// TwinCAT 3 PLC project LoadBank_Controller
// ProgramVersion: 3.1.4024.0
// libraries:
//   Tc2_Standard, * (Beckhoff Automation GmbH)
//   Tc2_System, * (Beckhoff Automation GmbH)
//   Tc2_Utilities, * (Beckhoff Automation GmbH)
//   Tc3_Module, * (Beckhoff Automation GmbH)
//   VisuSymbols,3.5.10.0,System
// project tree:
//   DUTs/ DUT_Alarm.TcDUT, DUT_Alarm_History_Record.TcDUT, DUT_Saved_Recipe.TcDUT, Recipe_Status.TcDUT, DUT_Emergency_Status.TcDUT, DUT_HMI_Step.TcDUT, DUT_Mode_Status.TcDUT, DUT_Recipe_Step.TcDUT, DUT_Simple_Config.TcDUT, DUT_Simple_Status.TcDUT
//   / GlobalTextList.TcGTLO, PlcTask.TcTTO, VisualizationManager.TcVMO (not stored), VISU_TASK.TcTTO
//   GVLs/ GVL_LoadBank_Constants.TcGVL, GVL_LoadBank_IO.TcGVL, GVL_LoadBank_Persistent.TcGVL, GVL_LoadBank_Runtime.TcGVL, GVL_Recipe_Storage.TcGVL
//   POUs/ FB_Auto_Mode.TcPOU, FB_DataLogger.TcPOU, FB_Gradual_Dump.TcPOU, FB_Alarm_Manager.TcPOU, FB_Load_Controller.TcPOU, FB_Maintenance_Mode.TcPOU, FB_Main_Contactor.TcPOU, FB_Manual_Mode.TcPOU, FB_Mode_Manager.TcPOU, FB_Numeric_Mode.TcPOU, FB_Recipe_Controller.TcPOU, FB_Recipe_Storage_Manager.TcPOU, FB_Reverse_Mode.TcPOU, FB_Single_Fan.TcPOU, FB_Temperature_Monitor.TcPOU, PRG_Main.TcPOU, PRG_Maint_Mode.TcPOU
// real-time tasks:
//   TASK PlcTask: cycle T#10ms, priority 20, ADS port 350
//   TASK VISU_TASK: cycle T#200000us, priority 30, ADS port 351

CONFIGURATION LoadBank_Controller
    RESOURCE PLC ON TwinCAT3
        TASK PlcTask(INTERVAL := T#10ms, PRIORITY := 20);
        TASK VISU_TASK(INTERVAL := T#200000us, PRIORITY := 30);
        PROGRAM PRG_Main WITH PlcTask : PRG_Main;
        PROGRAM VisuElems_Visu_Prg WITH VISU_TASK : VisuElems.Visu_Prg;
    END_RESOURCE
END_CONFIGURATION

// ---- DUTs/DUT_Alarm.TcDUT
// ============================================
// DUT_Alarm
// Structure for active alarm records
// ============================================

TYPE DUT_Alarm :
STRUCT
    ID                  : UINT;             // Alarm number (1-17)
    Name                : STRING(30);       // Short name "FAN FAULT"
    Description         : STRING(50);       // Detail "Motor overload tripped"
    Severity            : UINT;             // 1=Critical (Red), 2=Warning (Yellow)
    Active              : BOOL;             // Currently active?
    Acknowledged        : BOOL;             // Operator acknowledged?
    Timestamp_Occurred  : STRING(20);       // When alarm started
END_STRUCT
END_TYPE

// ---- DUTs/DUT_Alarm_History_Record.TcDUT
// ============================================
// DUT_Alarm_History_Record
// Structure for alarm history records
// ============================================

TYPE DUT_Alarm_History_Record :
STRUCT
    Alarm_ID            : UINT;             // Alarm number (1-17)
    Alarm_Name          : STRING(30);       // Short name
    Severity            : UINT;             // 1=Critical, 2=Warning
    Time_Occurred       : STRING(20);       // When alarm started
    Time_Cleared        : STRING(20);       // When alarm cleared
    Duration_Sec        : UDINT;            // How long active (seconds)
    Was_Acknowledged    : BOOL;             // Was it ack'd before clearing?
END_STRUCT
END_TYPE

// ---- DUTs/DUT_Saved_Recipe.TcDUT
// ============================================
// DATA TYPE: DUT_Saved_Recipe
// Add to your DUTs folder
// ============================================
TYPE DUT_Saved_Recipe :
STRUCT
    Recipe_Name             : STRING(40);       // Recipe display name
    Number_Of_Steps         : UINT;             // How many steps in this recipe
    Steps                   : ARRAY[1..20] OF DUT_Recipe_Step;  // The recipe steps
    Total_Duration          : TIME;             // Calculated total time
    Peak_Power_kW           : REAL;             // Calculated peak power
    Is_Valid                : BOOL;             // TRUE if recipe slot contains valid data
END_STRUCT
END_TYPE

// ---- DUTs/Recipe_Status.TcDUT
TYPE Recipe_Status :
STRUCT
    Recipe_Running          : BOOL;
    Recipe_Complete         : BOOL;
    Recipe_Aborted          : BOOL;
	Recipe_Paused 			: BOOL;
    Current_Step            : UINT;
    Current_Step_Name       : STRING(30);
    Current_Target_kW       : REAL;
    Step_Elapsed_Time       : TIME;
    Step_Remaining_Time     : TIME;
    Step_Duration           : TIME;
    Step_Progress_Pct       : REAL;
    Total_Recipe_Time       : TIME;
    Total_Elapsed_Time      : TIME;
    Total_Remaining_Time    : TIME;
    Recipe_Progress_Pct     : REAL;
    Status_Message          : STRING(100);
END_STRUCT
END_TYPE

// ---- DUTs/DUT_Emergency_Status.TcDUT
TYPE DUT_Emergency_Status :
STRUCT
    Emergency_Active        : BOOL;
    Emergency_Type          : STRING(20);
    Emergency_Complete      : BOOL;
    Ramp_Progress_Percent   : UINT;
    Status_Message          : STRING(100);
END_STRUCT
END_TYPE

// ---- DUTs/DUT_HMI_Step.TcDUT
TYPE DUT_HMI_Step :
STRUCT
    Step_Number             : UINT;
    Rated_Power_kW          : REAL;
    Status_Active           : BOOL;
    Status_Quarantined      : BOOL;
    Status_Feedback_Fault   : BOOL;
    Status_Power_Fault      : BOOL;
    Cycle_Count             : UDINT;
    Measured_Power_kW       : REAL;
    Power_Error_Percent     : REAL;
	Has_Feedback            : BOOL;
END_STRUCT
END_TYPE

// ---- DUTs/DUT_Mode_Status.TcDUT
TYPE DUT_Mode_Status :
STRUCT
    Active_Mode             : UINT;
    Mode_Name               : STRING(30);
    Mode_Ready              : BOOL;
    Mode_Transitioning      : BOOL;
    Status_Message          : STRING(100);
END_STRUCT
END_TYPE

// ---- DUTs/DUT_Recipe_Step.TcDUT
TYPE DUT_Recipe_Step :
STRUCT
    Step_Name               : STRING(40);
    Target_Power_kW         : REAL;
    Duration                : TIME;
    Enabled                 : BOOL := TRUE;
END_STRUCT
END_TYPE

// ---- DUTs/DUT_Simple_Config.TcDUT
TYPE DUT_Simple_Config :
STRUCT
    Number_Of_Steps         : UINT := 10;
    Number_Of_TCs           : UINT := 5;
    Rated_Voltage           : REAL := 480.0;
    Voltage_Name            : STRING(20) := '480V 3-Phase';
    Voltage_Tolerance       : REAL := 5.0;
    Step_Power              : ARRAY[1..100] OF REAL;
    Temp_Warning            : REAL := 80.0;
    Temp_Maximum            : REAL := 100.0;
    Temp_Critical           : REAL := 120.0;
    Temp_Dump_Rate          : REAL := 10.0;
    Fan_Pressurize_Time     : TIME := T#5s;
    Fan_Cooldown_Time       : TIME := T#30s;
    EStop_Controlled_Percent: REAL := 10.0;
    EStop_Controlled_Time   : TIME := T#1s;
    Auto_Level_Deadband     : REAL := 5.0;
    Step_Change_Delay       : TIME := T#500ms;
    Feedback_Timeout        : TIME := T#3s;
    Enable_Power_Monitoring : BOOL := TRUE;
    Power_Tolerance_Percent : REAL := 5.0;
    Power_Monitor_Delay     : TIME := T#10s;
END_STRUCT
END_TYPE

// ---- DUTs/DUT_Simple_Status.TcDUT
TYPE DUT_Simple_Status :
STRUCT
    Released_Power_kW       : REAL;
    Available_Power_kW      : REAL;
    Rated_Total_kW          : REAL;
    Power_Error_kW          : REAL;
    Active_Steps            : UINT;
    Quarantined_Steps       : UINT;
    Fan_Running             : BOOL;
    Fan_Fault               : BOOL;
    Fan_Cycle_Count         : UDINT;
    Temperature_Outlet_Avg  : REAL;
    Temperature_Outlet_Max  : REAL;
    Temperature_Inlet       : REAL;
    Temperature_DeltaT      : REAL;
    Hottest_TC_Number       : UINT;
    Voltage_L1_L2           : REAL;
    Voltage_L2_L3           : REAL;
    Voltage_L3_L1           : REAL;
    Voltage_Average         : REAL;
    Voltage_Imbalance       : REAL;
    Voltage_OK              : BOOL;
    Current_L1              : REAL;
    Current_L2              : REAL;
    Current_L3              : REAL;
    Current_Total           : REAL;
    Current_Imbalance       : REAL;
    System_Running          : BOOL;
    System_Ready            : BOOL;
    System_Fault            : BOOL;
    System_Warning          : BOOL;
    Emergency_Active        : BOOL;
    Temperature_Dump        : BOOL;
    Active_Mode             : UINT;
    Mode_Name               : STRING(30);
    Mode_Ready              : BOOL;
END_STRUCT
END_TYPE

// ---- GVLs/GVL_LoadBank_Constants.TcGVL
VAR_GLOBAL CONSTANT

    // ============================================
    // OPERATING MODES (ID numbers only)
    // ============================================
    LB_MODE_OFF             : UINT := 0;
    LB_MODE_AUTO_LEVELING   : UINT := 1;
    LB_MODE_NUMERIC    		: UINT := 2;
    LB_MODE_REVERSE_POWER   : UINT := 3;
    LB_MODE_MANUAL			: UINT := 4;
    LB_MODE_RECIPE          : UINT := 5;
    LB_MODE_MAINTENANCE     : UINT := 6;

    // ============================================
    // HARDWARE CONFIGURATION (Change per job)
    // ============================================
    LB_NUMBER_OF_STEPS      : UINT := 10;
    LB_NUMBER_OF_TCS        : UINT := 2;
    
    // ============================================
    // VOLTAGE CONFIGURATION
    // ============================================
    LB_VOLTAGE              : REAL := 480.0;
    LB_VOLTAGE_NAME         : STRING(20) := '480V 3-Phase';

    // ============================================
    // STEP POWER RATINGS (kW per step)
    // When you change LB_NUMBER_OF_STEPS, update this array to match
    // ============================================
    LB_STEP_POWER           : ARRAY[1..LB_NUMBER_OF_STEPS] OF REAL := [
        40.0, 40.0, 80.0, 80.0, 160.0, 160.0, 320.0, 320.0, 640.0, 640.0
    ];

    // ============================================
    // ARRAY LIMITS
    // ============================================
    LB_MAX_RECIPE_STEPS     : UINT := 20;
    LB_TREND_BUFFER_MAX     : UINT := 3600;
	
	// Manual Mode Switch Configuration
    LB_MANUAL_SWITCH_POWER      : ARRAY[1..8] OF REAL := [50.0, 100.0, 150.0, 200.0, 250.0, 300.0, 350.0, 400.0];
    LB_NUMBER_OF_SWITCHES       : USINT := 8;

END_VAR

// ---- GVLs/GVL_LoadBank_IO.TcGVL
VAR_GLOBAL

    // ============================================
    // EMERGENCY INPUTS (NC contacts)
    // TRUE = OK, FALSE = E-STOP PRESSED
    // ============================================
    IO_Emergency_Immediate      : BOOL;
    IO_Emergency_Controlled     : BOOL;

    // ============================================
    // MASTER ENABLE INPUT (Optional physical switch)
    // Only used when LB_ENABLE_PHYSICAL_MASTER = TRUE
    // ============================================
    IO_Physical_Master_Enable   : BOOL;

    // ============================================
    // FAN INPUTS
    // ============================================
    IO_Fan_Contactor_FB         : BOOL;             // NO: TRUE = contactor closed
    IO_Fan_Motor_Overload_OK    : BOOL;             // NC: TRUE = healthy, FALSE = FAULT
    IO_Fan_Pressure_OK          : BOOL;             // NO: TRUE = pressure OK

    // ============================================
    // MAIN CONTACTOR INPUT
    // ============================================
    IO_Main_Contactor_FB        : BOOL;             // NO: TRUE = contactor closed, load contactor

    // ============================================
    // LOAD STEP INPUTS
    // ============================================
    IO_Load_Contactor_FB        : ARRAY[1..LB_NUMBER_OF_STEPS] OF BOOL;     // NO: TRUE = closed
    IO_Step_Power               : ARRAY[1..LB_NUMBER_OF_STEPS] OF REAL;     // kW per step

    // ============================================
    // TEMPERATURE INPUTS
    // ============================================
    IO_Temperature_TC           : ARRAY[1..LB_NUMBER_OF_TCS] OF REAL;
    IO_Temperature_Inlet        : REAL;

    // ============================================
    // POWER METER INPUTS - VOLTAGE
    // ============================================
    IO_Voltage_L1_L2            : REAL;
    IO_Voltage_L2_L3            : REAL;
    IO_Voltage_L3_L1            : REAL;
    IO_Voltage_Average          : REAL;
    
    IO_Voltage_L1_LN            : REAL;
    IO_Voltage_L2_LN            : REAL;
    IO_Voltage_L3_LN            : REAL;

    // ============================================
    // POWER METER INPUTS - CURRENT
    // ============================================
    IO_Current_L1               : REAL;
    IO_Current_L2               : REAL;
    IO_Current_L3               : REAL;

    // ============================================
    // POWER METER INPUTS - SYSTEM
    // ============================================
    IO_Frequency                : REAL;
    IO_Power_Factor             : REAL;
    IO_Total_Power_kW           : REAL;
    IO_Total_Power_kVAR         : REAL;
    IO_Total_Power_kVA          : REAL;

    // ============================================
    // EXTERNAL POWER INPUT (Auto/Reverse modes)
    // ============================================
    IO_External_Power_kW        : REAL;

    // ============================================
    // DIGITAL OUTPUTS - CONTACTORS
    // ============================================
    IO_Fan_Contactor_Coil       : BOOL;
    IO_Main_Contactor_Coil      : BOOL;
    IO_Load_Contactor_Coil      : ARRAY[1..LB_NUMBER_OF_STEPS] OF BOOL;

    // ============================================
    // DIGITAL OUTPUTS - LED INDICATORS
    // ============================================
    IO_LED_General_Alarm        : BOOL;             // Red LED
    IO_LED_Warning              : BOOL;             // Yellow LED
    IO_LED_System_Normal        : BOOL;             // Green LED
	
	// ============================================
    // FAN PHYSICAL CONTROL (Optional)
    // Only used when LB_ENABLE_PHYSICAL_FAN = TRUE
    // ============================================
    IO_Physical_Fan_Start       : BOOL;             // Physical start button

END_VAR

// ---- GVLs/GVL_LoadBank_Persistent.TcGVL
// ============================================
// GVL_LoadBank_Persistent
// UPDATED: Separate EMG and TEMP dump settings
// ============================================

VAR_GLOBAL PERSISTENT

    // ============================================
    // TEMPERATURE CONFIG (ENG Page)
    // ============================================
    LB_OUTLET_WARNING_TEMP      : REAL := 350.0;
    LB_OUTLET_MAXIMUM_TEMP      : REAL := 400.0;
    LB_TC_OPEN_LIMIT            : REAL := 700.0;
    LB_TC_SHORT_LIMIT           : REAL := -50.0;
    
    LB_INLET_WARNING_TEMP       : REAL := 50.0;
    LB_INLET_MAXIMUM_TEMP       : REAL := 75.0;
    LB_INLET_TC_ENABLED         : BOOL := TRUE;

    // ============================================
    // FAN CONTROL (ENG Page)
    // ============================================
    LB_FAN_PRESSURIZE_TIME      : TIME := T#5s;
    LB_FAN_COOLDOWN_TIME        : TIME := T#180s;    // CHANGED: Was T#30s, now 3 min for normal/temp cooldown
    LB_FAN_FEEDBACK_TIMEOUT     : TIME := T#3s;
    LB_FAN_POST_DUMP_DELAY      : TIME := T#5s;      // CHANGED: Was T#3s, delay after EMG dump before fan stops
    LB_ENABLE_PHYSICAL_FAN      : BOOL := FALSE;

    // ============================================
    // MAIN CONTACTOR (ENG Page)
    // ============================================
    LB_MAIN_CONTACTOR_FB_TIMEOUT : TIME := T#3s;

    // ============================================
    // CONTROLLED EMERGENCY DUMP (ENG Page)
    // Fan uses short delay (LB_FAN_POST_DUMP_DELAY) after dump
    // ============================================
    LB_EMG_DUMP_PERCENT         : REAL := 10.0;     // NEW: % per step for EMG
    LB_EMG_DUMP_STEP_TIME       : TIME := T#1s;     // NEW: Time between steps for EMG

    // ============================================
    // OVER TEMPERATURE DUMP (ENG Page)
    // Fan uses full cooldown (LB_FAN_COOLDOWN_TIME) after dump
    // ============================================
    LB_TEMP_DUMP_PERCENT        : REAL := 10.0;     // NEW: % per step for temp
    LB_TEMP_DUMP_STEP_TIME      : TIME := T#2s;     // NEW: Time between steps for temp

    // ============================================
    // DUMP TIMEOUT (ENG Page)
    // ============================================
    LB_DUMP_TIMEOUT             : TIME := T#30s;    // KEPT: Safety timeout for any dump

    // ============================================
    // LOAD CONTROL
    // ============================================
    LB_AUTO_LEVEL_DEADBAND      : REAL := 5.0;
    LB_AUTO_LEVEL_HYSTERESIS    : REAL := 2.0;
    LB_STEP_UP_DELAY            : TIME := T#500ms;
    LB_STEP_DOWN_DELAY          : TIME := T#500ms;

    // ============================================
    // FEEDBACK MONITORING (ENG Page)
    // ============================================
    LB_ENABLE_FEEDBACK_MONITORING : BOOL := FALSE;
    LB_FEEDBACK_TIMEOUT           : TIME := T#3s;

    // ============================================
    // POWER MONITORING (ENG Page)
    // ============================================
    LB_ENABLE_POWER_MONITORING  : BOOL := FALSE;
    LB_POWER_TOLERANCE_PERCENT  : REAL := 5.0;
    LB_POWER_MONITOR_DELAY      : TIME := T#10s;

    // ============================================
    // VOLTAGE IMBALANCE (ENG Page)
    // ============================================
    LB_VOLTAGE_TOLERANCE        : REAL := 5.0;
    LB_V_IMBALANCE_WARNING      : REAL := 1.0;
    LB_V_IMBALANCE_CRITICAL     : REAL := 2.0;

    // ============================================
    // CURRENT IMBALANCE (ENG Page)
    // ============================================
    LB_I_IMBALANCE_WARNING      : REAL := 1.0;
    LB_I_IMBALANCE_CRITICAL     : REAL := 2.0;

    // ============================================
    // DATA LOGGER (ENG Page)
    // ============================================
    LB_LOG_ENABLE               : BOOL := TRUE;
    LB_USB_LOG_ENABLE           : BOOL := TRUE;
    LB_LOG_SAMPLE_TIME          : TIME := T#10s;
    LB_TREND_BUFFER_SIZE        : UINT := 360;
    LB_USB_LOG_PATH             : STRING(100) := 'C:\DataLog\';

    // ============================================
    // HMI DISPLAY CONFIG (ENG Page)
    // ============================================
    LB_HMI_Config_Mode_Auto     : BOOL := TRUE;
    LB_HMI_Config_Mode_Reverse  : BOOL := FALSE;
    LB_HMI_Config_Mode_Manual   : BOOL := FALSE;

    // ============================================
    // HMI THEME (Customer Page)
    // ============================================
    LB_HMI_Dark_Mode            : BOOL := FALSE;

    // ============================================
    // MAINTENANCE (Customer Page)
    // ============================================
    LB_Maint_Test_Duration_Sec  : INT := 30;
    
    // ============================================
    // MASTER ENABLE CONFIG (ENG Page)
    // ============================================
    LB_ENABLE_PHYSICAL_MASTER   : BOOL := FALSE;
    
    // ============================================
    // Engineer Login Credentials
    // ============================================
    HMI_Eng_Username        : STRING(20) := 'eng';
    HMI_Eng_Password        : STRING(20) := 'loadbank2025';
    HMI_Eng_Timeout_Min     : INT := 10;
	
	// Settings
	Maint_Mode_Power_Tolerance_Percent  : REAL := 10.0;
	Maint_Mode_Feedback_Timeout_ms      : INT := 2000;
	Maint_Mode_Test_Duration_Sec        : INT := 5;

END_VAR

// ---- GVLs/GVL_LoadBank_Runtime.TcGVL
// ============================================
// GVL_LoadBank_Runtime
// UPDATED: Added HMI status text variables
// ============================================

VAR_GLOBAL

    // ============================================
    // MASTER ENABLE CONTROL
    // ============================================
    HMI_Master_Enable           : BOOL;
    Master_Enable               : BOOL;
    Master_Enable_Blocked       : BOOL;
    Master_Enable_Was_Off       : BOOL;

    // ============================================
    // FAN START CONTROL
    // ============================================
    HMI_Fan_Start               : BOOL;
    Fan_Start_Command           : BOOL;
    Fan_Start_Blocked           : BOOL;
    Fan_Start_Was_Off           : BOOL;

    // ============================================
    // HMI MODE INPUTS
    // ============================================
    HMI_Mode_Select             : UINT;
    HMI_Target_Power_kW         : REAL;
    HMI_Target_Frequency        : REAL := 60.0;
    HMI_Target_Reverse_kW       : REAL;
    HMI_Recipe_Start            : BOOL;
    HMI_Recipe_Stop             : BOOL;
    HMI_Recipe_Pause            : BOOL;
    HMI_Manual_Step_Cmd         : ARRAY[1..LB_NUMBER_OF_STEPS] OF BOOL;
    HMI_Reset_Cmd               : BOOL;
    
    // ============================================
    // NUMERIC MODE HMI
    // ============================================
    Numeric_Mode_Status         : STRING(100);

    // ============================================
    // AUTO MODE HMI
    // ============================================
    HMI_Min_Load_kW             : REAL;
    Auto_Mode_Power_Error       : REAL;
    Auto_Mode_Status            : STRING(100);

    // ============================================
    // QUARANTINE CONTROL
    // ============================================
    Step_Quarantined            : ARRAY[1..LB_NUMBER_OF_STEPS] OF BOOL;
    Step_Quarantine_Feedback    : ARRAY[1..LB_NUMBER_OF_STEPS] OF BOOL;
    Step_Quarantine_Manual      : ARRAY[1..LB_NUMBER_OF_STEPS] OF BOOL;
    Step_Unquarantine_Cmd       : ARRAY[1..LB_NUMBER_OF_STEPS] OF BOOL;
    Step_Cycle_Count            : ARRAY[1..LB_NUMBER_OF_STEPS] OF UDINT;

    // ============================================
    // DUMP STATUS
    // ============================================
    Dump_Active                 : BOOL;
    Dump_Percent                : REAL := 100.0;
    Dump_Complete               : BOOL;
    Is_Temperature_Dump         : BOOL;
    Is_Emergency_Dump           : BOOL;

    // ============================================
    // MAIN CONTACTOR STATUS
    // ============================================
    Main_Contactor_Closed       : BOOL;
    Main_Contactor_Fault        : BOOL;
    Main_Contactor_Allowed      : BOOL;

    // ============================================
    // SYSTEM STATUS FLAGS
    // ============================================
    System_Ready                : BOOL;
    System_Running              : BOOL;
    System_Fault                : BOOL;

    // ============================================
    // ALARM STATUS
    // ============================================
    General_Alarm               : BOOL;
    General_Warning             : BOOL;
    System_Normal               : BOOL;
    Any_Fault_Active            : BOOL;

    // ============================================
    // ALARM COMMANDS (from HMI)
    // ============================================
    Alarm_Acknowledge_Cmd       : BOOL;
    Alarm_Reset_Cmd             : BOOL;

    // ============================================
    // STATUS TEXT (for HMI display)
    // ============================================
    Status_Fan                  : STRING(100);
    Status_Temperature          : STRING(100);
    Status_Main_Contactor       : STRING(100);
    Status_Load                 : STRING(100);
    Status_Dump                 : STRING(100);

    // ============================================
    // HMI STATUS BAR TEXT (NEW)
    // ============================================
    HMI_System_Status_Text      : STRING(100);      // NEW: Main status message for HMI status bar
    HMI_Alarm_Detail_Text       : STRING(100);      // NEW: Secondary detail message for HMI

    // ============================================
    // MODE CONTROL
    // ============================================
    Mode_Current                : UINT;
    Mode_Requested              : UINT;
    Mode_Target_Power           : REAL;

    // ============================================
    // IMBALANCE CALCULATIONS
    // ============================================
    Voltage_Imbalance_Percent   : REAL;
    Current_Imbalance_Percent   : REAL;
    Voltage_Imbalance_Warning   : BOOL;
    Voltage_Imbalance_Critical  : BOOL;
    Current_Imbalance_Warning   : BOOL;
    Current_Imbalance_Critical  : BOOL;

    // ============================================
    // TREND BUFFERS (for HMI)
    // ============================================
    Trend_Power_Released        : ARRAY[1..LB_TREND_BUFFER_MAX] OF REAL;
    Trend_Power_Target          : ARRAY[1..LB_TREND_BUFFER_MAX] OF REAL;
    Trend_Temp_TC1              : ARRAY[1..LB_TREND_BUFFER_MAX] OF REAL;
    Trend_Temp_TC2              : ARRAY[1..LB_TREND_BUFFER_MAX] OF REAL;
    Trend_Temp_TC3              : ARRAY[1..LB_TREND_BUFFER_MAX] OF REAL;
    Trend_Temp_TC4              : ARRAY[1..LB_TREND_BUFFER_MAX] OF REAL;
    Trend_Voltage_L1L2          : ARRAY[1..LB_TREND_BUFFER_MAX] OF REAL;
    Trend_Voltage_L2L3          : ARRAY[1..LB_TREND_BUFFER_MAX] OF REAL;
    Trend_Voltage_L3L1          : ARRAY[1..LB_TREND_BUFFER_MAX] OF REAL;
    Trend_Current_I1            : ARRAY[1..LB_TREND_BUFFER_MAX] OF REAL;
    Trend_Current_I2            : ARRAY[1..LB_TREND_BUFFER_MAX] OF REAL;
    Trend_Current_I3            : ARRAY[1..LB_TREND_BUFFER_MAX] OF REAL;
    Trend_Index                 : UINT;
    Trend_Sample_Count          : UINT;

    // ============================================
    // SYSTEM STATUS STRUCT (for HMI)
    // ============================================
    LB_System_Status            : DUT_Simple_Status;
    LB_Mode_Status              : DUT_Mode_Status;
    LB_Emergency_Status         : DUT_Emergency_Status;
    LB_Recipe_Status            : Recipe_Status;

    // ============================================
    // STEP STATUS (for HMI)
    // ============================================
    LB_HMI_Steps                : ARRAY[1..LB_NUMBER_OF_STEPS] OF DUT_HMI_Step;
    LB_RATED_KW                 : ARRAY[1..LB_NUMBER_OF_STEPS] OF REAL;

    // ============================================
    // HMI HELPER VARIABLES
    // ============================================
    LB_HMI_Temperature_Status   : INT;
    LB_HMI_Fan_Status           : INT;
    LB_HMI_System_Status        : INT;
    LB_HMI_V_Imbalance_Status   : INT;
    LB_HMI_I_Imbalance_Status   : INT;

    LB_HMI_Released_Percent     : REAL;
    LB_HMI_Available_Percent    : REAL;

    LB_HMI_Active_Count         : INT;
    LB_HMI_Inactive_Count       : INT;
    LB_HMI_Quarantined_Count    : INT;
    LB_HMI_Total_Steps          : INT;

    LB_HMI_Active_Bar_Width     : REAL;
    LB_HMI_Inactive_Bar_Width   : REAL;
    LB_HMI_Quarantine_Bar_Width : REAL;

    LB_HMI_Hottest_TC           : INT;
    LB_HMI_Mode_Text            : STRING(20);
    LB_HMI_Mode_Ready           : BOOL;
    LB_HMI_Emergency_Text       : STRING(30);
    
    // ============================================
    // MANUAL MODE HMI (8 Switches)
    // ============================================
    HMI_Manual_Switch           : ARRAY[1..8] OF BOOL;
    HMI_Manual_Selected_kW      : REAL;
    Manual_Mode_Status          : STRING(100);
    
    // ============================================
    // RECIPE MODE HMI 
    // ============================================
    HMI_Recipe_Number_Of_Steps  : UINT := 5;
    HMI_Recipe_Steps            : ARRAY[1..20] OF DUT_Recipe_Step;
    
    // ============================================
    // REVERSE MODE HMI
    // ============================================
    HMI_Follow_Percentage       : REAL := 100.0;
    Reverse_Mode_Target_Power   : REAL;
    Reverse_Mode_Status         : STRING(100);
	
	// ============================================
    // ALARM MANAGER OUTPUTS (from FB_Alarm_Manager)
    // ============================================
    LB_Alarm_List               : ARRAY[1..20] OF DUT_Alarm;        // Active alarm list for HMI
    LB_Alarm_List_Count         : UINT;                              // Number of active alarms
    LB_Alarm_History            : ARRAY[1..50] OF DUT_Alarm_History_Record;  // History buffer
    LB_Alarm_History_Count      : UINT;                              // Number of history records
    
    LB_Critical_Alarm_Count     : UINT;                              // Critical alarm count
    LB_Warning_Count            : UINT;                              // Warning count
    LB_Total_Alarm_Count        : UINT;                              // Total active count
    LB_Unacknowledged_Count     : UINT;                              // Unacknowledged count
    
    LB_New_Alarm_Trigger        : BOOL;                              // Pulse for new alarm popup
    LB_Newest_Alarm_ID          : UINT;                              // ID of newest alarm
    LB_Newest_Alarm_Name        : STRING(30);                        // Name of newest alarm
    
    // ============================================
    // ALARM MANAGER COMMANDS (from HMI)
    // ============================================
    HMI_Alarm_Acknowledge       : ARRAY[1..20] OF BOOL;              // Acknowledge individual alarm
    HMI_Alarm_Acknowledge_All   : BOOL;                              // Acknowledge all alarms
    HMI_Alarm_Clear_History     : BOOL;                              // Clear history buffer
	
	// ============================================
// MAINTENANCE MODE HMI
// ============================================
// Commands (from HMI buttons)
Maint_Mode_Toggle_Fan               : BOOL;
Maint_Mode_Toggle_Step              : BOOL;
Maint_Mode_Reset_Test               : BOOL;
Maint_Mode_Selected_Step            : INT := 1;
Maint_Mode_Self_Test_Start          : BOOL;
Maint_Mode_Self_Test_Stop           : BOOL;


// Status (to HMI display)
Maint_Mode_Feedback_Match           : BOOL;
Maint_Mode_Response_Time_ms         : INT;
Maint_Mode_Power_Within_Tolerance   : BOOL;
Maint_Mode_Self_Test_Running        : BOOL;
Maint_Mode_Self_Test_Current_Step   : INT;
Maint_Mode_Self_Test_Pass_Count     : INT;
Maint_Mode_Self_Test_Fail_Count     : INT;
Maint_Mode_Self_Test_Complete       : BOOL;
Maint_Mode_Timeout_Error_Count      : INT;
Maint_Mode_Self_Test_Timer_Sec      : INT;

END_VAR

// ---- GVLs/GVL_Recipe_Storage.TcGVL
VAR_GLOBAL PERSISTENT
    // 4 recipe storage slots
    Saved_Recipes           : ARRAY[1..4] OF DUT_Saved_Recipe;
END_VAR

VAR_GLOBAL
    // HMI Interface - Recipe Management
    HMI_Recipe_Select_Index     : UINT := 1;        // Which slot is selected (1-4)
    HMI_Recipe_Save_Cmd         : BOOL;             // Trigger to save current recipe
    HMI_Recipe_Load_Cmd         : BOOL;             // Trigger to load selected recipe
    HMI_Recipe_Delete_Cmd       : BOOL;             // Trigger to delete selected recipe
    
    // Recipe names for dropdown (bind to HMI combobox)
    HMI_Recipe_Name_1           : STRING(40);
    HMI_Recipe_Name_2           : STRING(40);
    HMI_Recipe_Name_3           : STRING(40);
    HMI_Recipe_Name_4           : STRING(40);
    
    // Status feedback
    HMI_Recipe_Operation_Status : STRING(50);       // "Saved", "Loaded", "Deleted", "Error"
END_VAR

// ---- POUs/PRG_Main.TcPOU
PROGRAM PRG_Main
VAR
    // ============================================
    // FUNCTION BLOCK INSTANCES
    // ============================================
    Single_Fan              : FB_Single_Fan;
    Temperature_Monitor     : FB_Temperature_Monitor;
    Gradual_Dump            : FB_Gradual_Dump;
    Main_Contactor          : FB_Main_Contactor;
    Load_Controller         : FB_Load_Controller;
    Mode_Manager            : FB_Mode_Manager;
    DataLogger              : FB_DataLogger;
    Alarm_Manager           : FB_Alarm_Manager;     // NEW - Alarm Manager
    
    // Mode FBs
    Auto_Mode               : FB_Auto_Mode;
    Numeric_Mode            : FB_Numeric_Mode;
    Reverse_Mode            : FB_Reverse_Mode;
    Manual_Mode             : FB_Manual_Mode;
    Recipe_Controller       : FB_Recipe_Controller;
    Maintenance_Mode        : FB_Maintenance_Mode;
    
    // Recipe Storage
    Recipe_Storage          : FB_Recipe_Storage_Manager;
    
    // ============================================
    // EMERGENCY STOP (internal)
    // ============================================
    EMG_Immediate_Active    : BOOL;
    EMG_Controlled_Active   : BOOL;
    Any_Emergency           : BOOL;
    
    // ============================================
    // ALARM RESET (internal)
    // ============================================
    Alarm_Reset_Combined    : BOOL;
    Alarm_Reset_Prev        : BOOL;
    Alarm_Reset_Pulse       : BOOL;
    
    // ============================================
    // INTERNAL
    // ============================================
    i                       : UINT;
    First_Scan              : BOOL := TRUE;
    
    // ============================================
    // FIX: Local TC buffer to convert [1..2] → [1..4]
    // ============================================
    Temp_TC_Buffer          : ARRAY[1..4] OF REAL;
END_VAR


// ============================================================
// FIRST SCAN INITIALIZATION
// ============================================================
IF First_Scan THEN
    HMI_Master_Enable := FALSE;
    HMI_Fan_Start := FALSE;
    Master_Enable_Was_Off := TRUE;
    Fan_Start_Was_Off := TRUE;
    First_Scan := FALSE;
END_IF;

// ============================================================
// EMERGENCY STOP DETECTION (NC contacts - TRUE = OK)
// ============================================================
EMG_Immediate_Active := NOT IO_Emergency_Immediate;
EMG_Controlled_Active := NOT IO_Emergency_Controlled;
Any_Emergency := EMG_Immediate_Active OR EMG_Controlled_Active;

// ============================================================
// ALARM RESET (rising edge detection)
// ============================================================
Alarm_Reset_Combined := Alarm_Reset_Cmd OR HMI_Reset_Cmd;
Alarm_Reset_Pulse := Alarm_Reset_Combined AND NOT Alarm_Reset_Prev;
Alarm_Reset_Prev := Alarm_Reset_Combined;

// Clear HMI reset command after processing
IF HMI_Reset_Cmd THEN
    HMI_Reset_Cmd := FALSE;
END_IF;

// ============================================================
// FIX: COPY TC READINGS INTO [1..4] BUFFER
// IO_Temperature_TC is [1..LB_NUMBER_OF_TCS] which is [1..2]
// FB_Temperature_Monitor expects [1..4]
// ============================================================
Temp_TC_Buffer[1] := IO_Temperature_TC[1];
Temp_TC_Buffer[2] := IO_Temperature_TC[2];
Temp_TC_Buffer[3] := 0.0;    // Not connected (only 2 TCs)
Temp_TC_Buffer[4] := 0.0;    // Not connected (only 2 TCs)

// ============================================================
// TEMPERATURE MONITOR
// FIX: Pass Temp_TC_Buffer [1..4] instead of IO_Temperature_TC [1..2]
// ============================================================
Temperature_Monitor(
    Outlet_TC_Readings := Temp_TC_Buffer,
    Inlet_TC_Reading := IO_Temperature_Inlet,
    Outlet_TC_Count := LB_NUMBER_OF_TCS,
    Inlet_TC_Enabled := LB_INLET_TC_ENABLED,
    Outlet_Warning_Temp := LB_OUTLET_WARNING_TEMP,
    Outlet_Maximum_Temp := LB_OUTLET_MAXIMUM_TEMP,
    TC_Open_Limit := LB_TC_OPEN_LIMIT,
    TC_Short_Limit := LB_TC_SHORT_LIMIT,
    Inlet_Warning_Temp := LB_INLET_WARNING_TEMP,
    Inlet_Maximum_Temp := LB_INLET_MAXIMUM_TEMP,
    Enable := TRUE,
    Reset := Alarm_Reset_Pulse
);

// Update status
Status_Temperature := Temperature_Monitor.Status_Text;
LB_System_Status.Temperature_Outlet_Avg := Temperature_Monitor.Outlet_Temp_Avg;
LB_System_Status.Temperature_Outlet_Max := Temperature_Monitor.Outlet_Temp_Max;
LB_System_Status.Temperature_Inlet := Temperature_Monitor.Inlet_Temp;
LB_System_Status.Temperature_DeltaT := Temperature_Monitor.Delta_T;
LB_System_Status.Hottest_TC_Number := Temperature_Monitor.Hottest_TC_Index;

// HMI temperature status
IF Temperature_Monitor.Any_Overtemp THEN
    LB_HMI_Temperature_Status := 2;     // Maximum
ELSIF Temperature_Monitor.Any_Warning THEN
    LB_HMI_Temperature_Status := 1;     // Warning
ELSE
    LB_HMI_Temperature_Status := 0;     // Normal
END_IF;

// ============================================================
// GRADUAL DUMP (UPDATED - Separate EMG and TEMP rates)
// ============================================================
Gradual_Dump(
    Temp_Dump_Trigger := Temperature_Monitor.Dump_Command,
    EMG_Dump_Trigger := EMG_Controlled_Active,
    Current_Power_kW := Load_Controller.Released_Power_kW,
    Rated_Power_kW := Load_Controller.Rated_Total_kW,
    EMG_Percent_Per_Step := LB_EMG_DUMP_PERCENT,
    EMG_Step_Time := LB_EMG_DUMP_STEP_TIME,
    Temp_Percent_Per_Step := LB_TEMP_DUMP_PERCENT,
    Temp_Step_Time := LB_TEMP_DUMP_STEP_TIME,
    Dump_Timeout := LB_DUMP_TIMEOUT,
    Enable := TRUE,
    Reset := Alarm_Reset_Pulse
);

// Update runtime variables
Dump_Active := Gradual_Dump.Dump_Active;
Dump_Complete := Gradual_Dump.Dump_Complete;
Dump_Percent := Gradual_Dump.Dump_Percent;
Is_Temperature_Dump := Gradual_Dump.Is_Temperature_Dump;
Is_Emergency_Dump := Gradual_Dump.Is_Emergency_Dump;
Status_Dump := Gradual_Dump.Status_Text;

// ============================================================
// ALARM MANAGER (NEW - Replaces inline alarm aggregation)
// ============================================================
Alarm_Manager(
    // Emergency
    IN_Emergency_Immediate := EMG_Immediate_Active,
    IN_Emergency_Controlled := EMG_Controlled_Active,
    
    // Temperature
    IN_Temp_Overtemp := Temperature_Monitor.Any_Overtemp,
    IN_Temp_Warning := Temperature_Monitor.Any_Warning,
    IN_TC_Sensor_Fail := Temperature_Monitor.TC_Fail_Dump_Required,
    IN_Inlet_Overtemp := Temperature_Monitor.Inlet_TC_Overtemp AND LB_INLET_TC_ENABLED,
    IN_Inlet_TC_Fail := Temperature_Monitor.Inlet_TC_Fail AND LB_INLET_TC_ENABLED,
    IN_TC_Contingency := Temperature_Monitor.Contingency_Mode,
    
    // Fan
    IN_Fan_Motor_Overload := Single_Fan.Fault_Motor_Overload,
    IN_Fan_Pressure_Fail := Single_Fan.Fault_Pressure,
    IN_Fan_Contactor_Fail := Single_Fan.Fault_Contactor,
    
    // Main Contactor
    IN_Main_Contactor_Fail := Main_Contactor.Contactor_Fault,
    
    // Load Controller
    IN_Step_Feedback_Fault := Load_Controller.Any_Feedback_Fault,
    IN_Power_Mismatch := Load_Controller.Total_Power_Warning,
    
    // Gradual Dump
    IN_Dump_Timeout := Gradual_Dump.Dump_Timeout_Fault,
    
    // Imbalance
    IN_Voltage_Imbalance := Voltage_Imbalance_Warning,
    IN_Current_Imbalance := Current_Imbalance_Warning,
    
    // RTC (connect if available, otherwise leave defaults)
    RTC_Valid := FALSE,     // Change to TRUE and connect RTC if you have one
    
    // Commands from HMI
    Acknowledge_Alarm := HMI_Alarm_Acknowledge,
    Acknowledge_All_Cmd := HMI_Alarm_Acknowledge_All,
    Reset_Cmd := Alarm_Reset_Pulse,
    Clear_History_Cmd := HMI_Alarm_Clear_History,
    
    Enable := TRUE
);

// Copy Alarm Manager outputs to GVL
General_Alarm := Alarm_Manager.General_Alarm;
General_Warning := Alarm_Manager.General_Warning;
System_Normal := Alarm_Manager.System_Normal;
Any_Fault_Active := Alarm_Manager.Any_Fault_Active;

// LED outputs
IO_LED_General_Alarm := Alarm_Manager.LED_Alarm;
IO_LED_Warning := Alarm_Manager.LED_Warning;
IO_LED_System_Normal := Alarm_Manager.LED_Normal;

// Alarm list and counts for HMI
LB_Alarm_List := Alarm_Manager.Alarm_List;
LB_Alarm_List_Count := Alarm_Manager.Alarm_List_Count;
LB_Alarm_History := Alarm_Manager.Alarm_History;
LB_Alarm_History_Count := Alarm_Manager.History_Count;

LB_Critical_Alarm_Count := Alarm_Manager.Critical_Alarm_Count;
LB_Warning_Count := Alarm_Manager.Warning_Count;
LB_Total_Alarm_Count := Alarm_Manager.Total_Active_Count;
LB_Unacknowledged_Count := Alarm_Manager.Unacknowledged_Count;

LB_New_Alarm_Trigger := Alarm_Manager.New_Alarm_Trigger;
LB_Newest_Alarm_ID := Alarm_Manager.Newest_Alarm_ID;
LB_Newest_Alarm_Name := Alarm_Manager.Newest_Alarm_Name;

// ============================================================
// MASTER ENABLE CONTROL
// ============================================================

// Force HMI off on ANY alarm
IF General_Alarm THEN
    HMI_Master_Enable := FALSE;
    Master_Enable_Blocked := TRUE;
END_IF;

// Physical button cycle tracking (must go OFF before ON after alarm)
IF LB_ENABLE_PHYSICAL_MASTER THEN
    // Track if physical was OFF
    IF NOT IO_Physical_Master_Enable THEN
        Master_Enable_Was_Off := TRUE;
    END_IF;
    
    // Clear block when cycled OFF after fault cleared
    IF NOT General_Alarm AND Master_Enable_Was_Off AND NOT IO_Physical_Master_Enable THEN
        Master_Enable_Blocked := FALSE;
    END_IF;
    
    // Reset tracking when turned ON
    IF IO_Physical_Master_Enable THEN
        Master_Enable_Was_Off := FALSE;
    END_IF;
    
    // Combine Master Enable sources
    Master_Enable := (HMI_Master_Enable OR IO_Physical_Master_Enable) 
                     AND NOT Master_Enable_Blocked
                     AND NOT General_Alarm;
ELSE
    // HMI only
    IF NOT General_Alarm AND Master_Enable_Was_Off THEN
        Master_Enable_Blocked := FALSE;
    END_IF;
    
    Master_Enable := HMI_Master_Enable AND NOT General_Alarm;
END_IF;

// ============================================================
// FAN CONTROL
// ============================================================

// Force HMI off on fan fault
IF Single_Fan.Fan_Fault THEN
    HMI_Fan_Start := FALSE;
    Fan_Start_Blocked := TRUE;
END_IF;

// Physical fan button cycle tracking
IF LB_ENABLE_PHYSICAL_FAN THEN
    IF NOT IO_Physical_Fan_Start THEN
        Fan_Start_Was_Off := TRUE;
    END_IF;
    
    IF NOT Single_Fan.Fan_Fault AND Fan_Start_Was_Off AND NOT IO_Physical_Fan_Start THEN
        Fan_Start_Blocked := FALSE;
    END_IF;
    
    IF IO_Physical_Fan_Start THEN
        Fan_Start_Was_Off := FALSE;
    END_IF;
    
    // Combine Fan Start sources
    Fan_Start_Command := (HMI_Fan_Start OR IO_Physical_Fan_Start)
                         AND NOT Fan_Start_Blocked;
ELSE
    IF NOT Single_Fan.Fan_Fault AND Fan_Start_Was_Off THEN
        Fan_Start_Blocked := FALSE;
    END_IF;
    
    Fan_Start_Command := HMI_Fan_Start AND NOT Fan_Start_Blocked;
END_IF;

// Call Single Fan FB (UPDATED - Added Is_Temperature_Dump)
Single_Fan(
    HMI_Start := HMI_Fan_Start,
    Physical_Start := IO_Physical_Fan_Start,
    Physical_Enabled := LB_ENABLE_PHYSICAL_FAN,
    Contactor_Feedback := IO_Fan_Contactor_FB,
    Motor_Overload_OK := IO_Fan_Motor_Overload_OK,
    Pressure_OK := IO_Fan_Pressure_OK,
    Emergency_Immediate := EMG_Immediate_Active,
    Emergency_Controlled := Is_Emergency_Dump,
    Is_Temperature_Dump := Is_Temperature_Dump,
    Dump_Complete := Dump_Complete,
    Pressurize_Time := LB_FAN_PRESSURIZE_TIME,
    Cooldown_Time := LB_FAN_COOLDOWN_TIME,
    Feedback_Timeout := LB_FAN_FEEDBACK_TIMEOUT,
    Post_Dump_Delay := LB_FAN_POST_DUMP_DELAY,
    Enable := Fan_Start_Command,
    Reset_Fault := Alarm_Reset_Pulse
);

// Fan output
IO_Fan_Contactor_Coil := Single_Fan.Contactor_Output;

// Update status
Status_Fan := Single_Fan.Status_Message;
LB_System_Status.Fan_Running := Single_Fan.Fan_Running;
LB_System_Status.Fan_Fault := Single_Fan.Fan_Fault;
LB_System_Status.Fan_Cycle_Count := Single_Fan.Cycle_Count;

// HMI fan status
IF Single_Fan.Fan_Fault THEN
    LB_HMI_Fan_Status := 5;         // Fault
ELSIF Single_Fan.Fan_Running AND Single_Fan.Fan_Pressurized THEN
    LB_HMI_Fan_Status := 3;         // Running
ELSIF Single_Fan.Fan_Running AND NOT Single_Fan.Fan_Pressurized THEN
    LB_HMI_Fan_Status := 2;         // Pressurizing
ELSIF Single_Fan.Contactor_Output THEN
    LB_HMI_Fan_Status := 1;         // Starting
ELSE
    LB_HMI_Fan_Status := 0;         // Off
END_IF;

// ============================================================
// MAIN CONTACTOR
// ============================================================
Main_Contactor(
    Master_Enable := Master_Enable,
    Fan_Running := Single_Fan.Fan_Running,
    Fan_Pressurized := Single_Fan.Fan_Pressurized,
    Any_Alarm := General_Alarm,
    Dump_Active := Dump_Active,
    Dump_Complete := Dump_Complete,
    Is_Temperature_Dump := Is_Temperature_Dump,
    Contactor_Feedback := IO_Main_Contactor_FB,
    Feedback_Timeout := LB_MAIN_CONTACTOR_FB_TIMEOUT,
    Enable := TRUE,
    Reset := Alarm_Reset_Pulse
);

// Main contactor output
IO_Main_Contactor_Coil := Main_Contactor.Contactor_Output;

// Update status
Main_Contactor_Closed := Main_Contactor.Contactor_Closed;
Main_Contactor_Fault := Main_Contactor.Contactor_Fault;
Main_Contactor_Allowed := Main_Contactor.Contactor_Output;
Status_Main_Contactor := Main_Contactor.Status_Text;

// ============================================================
// SYSTEM STATUS
// ============================================================
System_Ready := Single_Fan.Fan_Running 
                AND Single_Fan.Fan_Pressurized 
                AND NOT General_Alarm
                AND Master_Enable;

System_Running := Main_Contactor_Closed 
                  AND Load_Controller.Active_Step_Count > 0;

System_Fault := General_Alarm;

LB_System_Status.System_Ready := System_Ready;
LB_System_Status.System_Running := System_Running;
LB_System_Status.System_Fault := System_Fault;

// HMI system status
IF System_Fault THEN
    LB_HMI_System_Status := 3;      // Fault
ELSIF System_Running THEN
    LB_HMI_System_Status := 2;      // Running
ELSIF System_Ready THEN
    LB_HMI_System_Status := 1;      // Ready
ELSE
    LB_HMI_System_Status := 0;      // Off
END_IF;

// ============================================================
// MODE MANAGER
// ============================================================
Mode_Manager(
    Mode_Select := HMI_Mode_Select,
    Master_Enable := Master_Enable,
    Emergency_Active := Any_Emergency,
    System_Ready := System_Ready
);

// Update status
Mode_Current := Mode_Manager.Active_Mode;
LB_HMI_Mode_Text := Mode_Manager.Mode_Name;
LB_HMI_Mode_Ready := Mode_Manager.Mode_Ready;

// ============================================================
// MODE EXECUTION - GET TARGET POWER
// ============================================================
Mode_Target_Power := 0.0;

CASE Mode_Manager.Active_Mode OF

    LB_MODE_OFF:
        Mode_Target_Power := 0.0;
        
    LB_MODE_AUTO_LEVELING:
        Auto_Mode(
            Mode_Active := TRUE,
            External_Power_kW := IO_External_Power_kW,
            Min_Load_kW := HMI_Min_Load_kW,
            Available_Power_kW := Load_Controller.Available_Power_kW,
            Deadband_kW := LB_AUTO_LEVEL_DEADBAND,
            System_Ready := System_Ready
        );
        Mode_Target_Power := Auto_Mode.Target_Power_kW;
        
        // Copy to GVL for HMI
        Auto_Mode_Power_Error := Auto_Mode.Power_Error;
        Auto_Mode_Status := Auto_Mode.Status_Text;
        
    LB_MODE_NUMERIC:
        Numeric_Mode(
            Mode_Active := TRUE,
            Target_Power_Setpoint := HMI_Target_Power_kW,
            Rated_Power_kW := Load_Controller.Rated_Total_kW,
            System_Ready := System_Ready
        );
        Mode_Target_Power := Numeric_Mode.Target_Power_kW;
        
        // Copy to GVL for HMI
        Numeric_Mode_Status := Numeric_Mode.Status_Text;
        
    LB_MODE_REVERSE_POWER:
        Reverse_Mode(
            Mode_Active := TRUE,
            Generator_Power_kW := IO_External_Power_kW,
            Follow_Percentage := HMI_Follow_Percentage,
            Max_Power_kW := Load_Controller.Available_Power_kW,
            System_Ready := System_Ready
        );
        Mode_Target_Power := Reverse_Mode.Target_Power_kW;
        
        // Copy to GVL for HMI
        Reverse_Mode_Target_Power := Reverse_Mode.Target_Power_kW;
        Reverse_Mode_Status := Reverse_Mode.Status_Text;

    LB_MODE_MANUAL:
        Manual_Mode(
            Number_Of_Switches := LB_NUMBER_OF_SWITCHES,
            Switch_Status := HMI_Manual_Switch,
            Switch_Power := LB_MANUAL_SWITCH_POWER
        );
        Mode_Target_Power := Manual_Mode.Target_Power_kW;
        
        HMI_Manual_Selected_kW := Manual_Mode.Target_Power_kW;
        
        IF Mode_Target_Power > 0 THEN
            Manual_Mode_Status := 'Manual control active';
        ELSE
            Manual_Mode_Status := 'Select switches to apply load';
        END_IF;
        
    LB_MODE_RECIPE:
        Recipe_Controller(
            Recipe_Enable := Master_Enable,
            Recipe_Start := HMI_Recipe_Start,
            Recipe_Pause := HMI_Recipe_Pause,
            Recipe_Abort := HMI_Recipe_Stop,
            Recipe_Steps := HMI_Recipe_Steps,
            Number_Of_Steps := HMI_Recipe_Number_Of_Steps,
            Current_Power_kW := LB_System_Status.Released_Power_kW
        );
        Mode_Target_Power := Recipe_Controller.Target_Power_kW;
        
        // Copy FB outputs to GVL for HMI
        LB_Recipe_Status.Recipe_Running := Recipe_Controller.Recipe_Running;
        LB_Recipe_Status.Recipe_Paused := Recipe_Controller.Recipe_Paused;
        LB_Recipe_Status.Recipe_Complete := Recipe_Controller.Recipe_Complete;
        LB_Recipe_Status.Recipe_Aborted := Recipe_Controller.Recipe_Aborted;
        LB_Recipe_Status.Current_Step := Recipe_Controller.Current_Step_Number;
        LB_Recipe_Status.Current_Step_Name := Recipe_Controller.Current_Step_Name;
        LB_Recipe_Status.Current_Target_kW := Recipe_Controller.Target_Power_kW;
        LB_Recipe_Status.Step_Elapsed_Time := Recipe_Controller.Step_Elapsed_Time;
        LB_Recipe_Status.Step_Remaining_Time := Recipe_Controller.Step_Remaining_Time;
        LB_Recipe_Status.Total_Recipe_Time := Recipe_Controller.Total_Recipe_Time;
        LB_Recipe_Status.Total_Elapsed_Time := Recipe_Controller.Total_Elapsed_Time;
        LB_Recipe_Status.Total_Remaining_Time := Recipe_Controller.Total_Remaining_Time;
        LB_Recipe_Status.Recipe_Progress_Pct := Recipe_Controller.Recipe_Progress_Percent;
        LB_Recipe_Status.Status_Message := Recipe_Controller.Status_Message;
        
    LB_MODE_MAINTENANCE:
        Maintenance_Mode(
            Mode_Active := TRUE,
            Master_Enable := Master_Enable,
            Emergency_Active := Any_Emergency
        );
        // Maintenance mode uses direct step control

END_CASE;

// ============================================================
// APPLY DUMP LIMIT TO TARGET
// ============================================================
IF Dump_Active OR Dump_Complete THEN
    Mode_Target_Power := Gradual_Dump.Target_Power_kW;
END_IF;

// ============================================================
// LOAD CONTROLLER
// ============================================================
Load_Controller(
    Target_Power_kW := Mode_Target_Power,
    Main_Contactor_Closed := Main_Contactor_Closed,
    Step_Power_Rating := LB_STEP_POWER,
    Number_Of_Steps := LB_NUMBER_OF_STEPS,
    Step_Feedback := IO_Load_Contactor_FB,
    Measured_Total_Power := IO_Total_Power_kW,
    Step_Quarantine_Manual := Step_Quarantine_Manual,
    Step_Unquarantine_Cmd := Step_Unquarantine_Cmd,
    Maintenance_Mode := (Mode_Manager.Active_Mode = LB_MODE_MAINTENANCE),
    Manual_Step_Cmd := HMI_Manual_Step_Cmd,
    Deadband_kW := LB_AUTO_LEVEL_DEADBAND,
    Step_Up_Delay := LB_STEP_UP_DELAY,
    Step_Down_Delay := LB_STEP_DOWN_DELAY,
    Feedback_Timeout := LB_FEEDBACK_TIMEOUT,
    Enable_Feedback_Monitoring := LB_ENABLE_FEEDBACK_MONITORING,
    Power_Tolerance_Percent := LB_POWER_TOLERANCE_PERCENT,
    Power_Monitor_Delay := LB_POWER_MONITOR_DELAY,
    Enable_Power_Monitoring := LB_ENABLE_POWER_MONITORING,
    Enable := Mode_Manager.Enable_Output,
    Reset := Alarm_Reset_Pulse
);

// Step coil outputs
FOR i := 1 TO LB_NUMBER_OF_STEPS DO
    IO_Load_Contactor_Coil[i] := Load_Controller.Step_Coil_Cmd[i];
END_FOR;

// Update status
Status_Load := Load_Controller.Status_Text;
LB_System_Status.Released_Power_kW := Load_Controller.Released_Power_kW;
LB_System_Status.Available_Power_kW := Load_Controller.Available_Power_kW;
LB_System_Status.Rated_Total_kW := Load_Controller.Rated_Total_kW;
LB_System_Status.Active_Steps := Load_Controller.Active_Step_Count;
LB_System_Status.Quarantined_Steps := Load_Controller.Quarantined_Step_Count;

// Copy to runtime variables
FOR i := 1 TO LB_NUMBER_OF_STEPS DO
    Step_Quarantined[i] := Load_Controller.Step_Quarantined[i];
    Step_Quarantine_Feedback[i] := Load_Controller.Step_Quarantine_Feedback[i];
    Step_Cycle_Count[i] := Load_Controller.Step_Cycle_Count[i];
END_FOR;

// HMI step counts
LB_HMI_Active_Count := UINT_TO_INT(Load_Controller.Active_Step_Count);
LB_HMI_Quarantined_Count := UINT_TO_INT(Load_Controller.Quarantined_Step_Count);
LB_HMI_Inactive_Count := UINT_TO_INT(LB_NUMBER_OF_STEPS) - LB_HMI_Active_Count - LB_HMI_Quarantined_Count;
LB_HMI_Total_Steps := UINT_TO_INT(LB_NUMBER_OF_STEPS);

// HMI power percentages
IF Load_Controller.Rated_Total_kW > 0.0 THEN
    LB_HMI_Released_Percent := (Load_Controller.Released_Power_kW / Load_Controller.Rated_Total_kW) * 100.0;
    LB_HMI_Available_Percent := (Load_Controller.Available_Power_kW / Load_Controller.Rated_Total_kW) * 100.0;
ELSE
    LB_HMI_Released_Percent := 0.0;
    LB_HMI_Available_Percent := 0.0;
END_IF;

// ============================================================
// CALCULATE BAR WIDTHS FOR HMI (3-segment steps bar)
// ============================================================
IF LB_HMI_Total_Steps > 0 THEN
    LB_HMI_Active_Bar_Width := (INT_TO_REAL(LB_HMI_Active_Count) / INT_TO_REAL(LB_HMI_Total_Steps)) * 343.0;
    LB_HMI_Quarantine_Bar_Width := (INT_TO_REAL(LB_HMI_Quarantined_Count) / INT_TO_REAL(LB_HMI_Total_Steps)) * 343.0;
    LB_HMI_Inactive_Bar_Width := (INT_TO_REAL(LB_HMI_Inactive_Count) / INT_TO_REAL(LB_HMI_Total_Steps)) * 343.0;
ELSE
    LB_HMI_Active_Bar_Width := 0.0;
    LB_HMI_Quarantine_Bar_Width := 0.0;
    LB_HMI_Inactive_Bar_Width := 0.0;
END_IF;

// ============================================================
// UPDATE HMI STEP ARRAY
// FIX: Use correct DUT_HMI_Step field names
// ============================================================
FOR i := 1 TO LB_NUMBER_OF_STEPS DO
    LB_HMI_Steps[i].Step_Number := i;
    LB_HMI_Steps[i].Rated_Power_kW := LB_STEP_POWER[i];
    LB_HMI_Steps[i].Status_Active := Load_Controller.Step_Coil_Cmd[i];
    LB_HMI_Steps[i].Status_Quarantined := Step_Quarantined[i];
    LB_HMI_Steps[i].Has_Feedback := IO_Load_Contactor_FB[i];
    LB_HMI_Steps[i].Cycle_Count := Step_Cycle_Count[i];
END_FOR;

// ============================================================
// DATA LOGGER
// FIX: Use Temp_TC_Buffer instead of IO_Temperature_TC[3]/[4]
// ============================================================
DataLogger(
    Enable := LB_LOG_ENABLE,
    USB_Log_Enable := LB_USB_LOG_ENABLE,
    Sample_Time := LB_LOG_SAMPLE_TIME,
    Buffer_Size := LB_TREND_BUFFER_SIZE,
    
    // Power inputs
    Power_Released := LB_System_Status.Released_Power_kW,
    Power_Target := Mode_Target_Power,
    
    // Temperature inputs - use buffer (always [1..4])
    Temp_TC1 := Temp_TC_Buffer[1],
    Temp_TC2 := Temp_TC_Buffer[2],
    Temp_TC3 := Temp_TC_Buffer[3],
    Temp_TC4 := Temp_TC_Buffer[4],
    Number_Of_TCs := LB_NUMBER_OF_TCS,
    
    // Voltage inputs
    Voltage_L1L2 := IO_Voltage_L1_L2,
    Voltage_L2L3 := IO_Voltage_L2_L3,
    Voltage_L3L1 := IO_Voltage_L3_L1,
    
    // Current inputs
    Current_I1 := IO_Current_L1,
    Current_I2 := IO_Current_L2,
    Current_I3 := IO_Current_L3,
    
    // USB path
    USB_Path := LB_USB_LOG_PATH
);

// ============================================================
// HOTTEST TC FOR HMI
// ============================================================
LB_HMI_Hottest_TC := UINT_TO_INT(Temperature_Monitor.Hottest_TC_Index);

// ============================================================
// HMI STATUS BAR TEXT (UPDATED - Uses Alarm_Manager + operational states)
// ============================================================

// When alarms are active, use Alarm_Manager status text
IF Alarm_Manager.Total_Active_Count > 0 THEN
    HMI_System_Status_Text := Alarm_Manager.Status_Text;
    HMI_Alarm_Detail_Text := Alarm_Manager.Detail_Text;
ELSE
    // No alarms - show operational status
    IF System_Running THEN
        HMI_System_Status_Text := 'RUNNING';
        HMI_Alarm_Detail_Text := LB_HMI_Mode_Text;
    ELSIF System_Ready THEN
        HMI_System_Status_Text := 'READY';
        HMI_Alarm_Detail_Text := 'Select mode to start';
    ELSIF Single_Fan.Fan_Running THEN
        HMI_System_Status_Text := 'FAN RUNNING';
        HMI_Alarm_Detail_Text := Status_Fan;
    ELSIF Single_Fan.Contactor_Output THEN
        HMI_System_Status_Text := 'FAN STARTING';
        HMI_Alarm_Detail_Text := Status_Fan;
    ELSE
        HMI_System_Status_Text := 'STOPPED';
        IF NOT HMI_Master_Enable THEN
            HMI_Alarm_Detail_Text := 'Enable master to start';
        ELSIF NOT HMI_Fan_Start THEN
            HMI_Alarm_Detail_Text := 'Start fan to continue';
        ELSE
            HMI_Alarm_Detail_Text := Status_Fan;
        END_IF;
    END_IF;
END_IF;

// Emergency text for header display
IF EMG_Immediate_Active THEN
    LB_HMI_Emergency_Text := 'IMMEDIATE E-STOP';
ELSIF EMG_Controlled_Active OR Is_Emergency_Dump THEN
    LB_HMI_Emergency_Text := 'CONTROLLED E-STOP';
ELSIF Is_Temperature_Dump THEN
    LB_HMI_Emergency_Text := 'OVER TEMPERATURE';
ELSE
    LB_HMI_Emergency_Text := '';
END_IF;

END_PROGRAM

// ---- POUs/FB_Single_Fan.TcPOU
FUNCTION_BLOCK FB_Single_Fan
// ============================================
// SINGLE FAN CONTROLLER
// UPDATED: Added Is_Temperature_Dump input
// - EMG dump: Short delay (Post_Dump_Delay) then fan OFF
// - TEMP dump: Full cooldown (Cooldown_Time) then fan OFF
// - Normal stop: Full cooldown (Cooldown_Time) then fan OFF
// ============================================

VAR_INPUT
    HMI_Start               : BOOL;             // HMI button (PLC forces OFF on fault)
    Physical_Start          : BOOL;             // Physical button (PLC cannot control)
    Physical_Enabled        : BOOL;             // TRUE = physical button required
    
    Contactor_Feedback      : BOOL;             // NO: TRUE = contactor closed
    Motor_Overload_OK       : BOOL;             // NC: TRUE = healthy, FALSE = FAULT
    Pressure_OK             : BOOL;             // NO: TRUE = pressure OK
    
    Emergency_Immediate     : BOOL;             // TRUE = Stop NOW (instant)
    Emergency_Controlled    : BOOL;             // TRUE = EMG Controlled stop active (short delay after dump)
    Is_Temperature_Dump     : BOOL;             // NEW: TRUE = Temp dump active (full cooldown after dump)
    Dump_Complete           : BOOL;             // TRUE = Load at 0%
    
    Pressurize_Time         : TIME := T#5s;
    Cooldown_Time           : TIME := T#180s;   // CHANGED: Default 3 min for normal/temp cooldown
    Feedback_Timeout        : TIME := T#3s;
    Post_Dump_Delay         : TIME := T#5s;     // CHANGED: Default 5 sec for EMG only
    
    Enable                  : BOOL;
    Reset_Fault             : BOOL;
END_VAR

VAR_OUTPUT
    Contactor_Output        : BOOL;
    Fan_Running             : BOOL;
    Fan_Pressurized         : BOOL;
    
    Fan_Fault               : BOOL;
    Fault_Motor_Overload    : BOOL;
    Fault_Pressure          : BOOL;
    Fault_Contactor         : BOOL;
    Fault_Emergency         : BOOL;
    
    Force_HMI_Off           : BOOL;             // TRUE = force HMI_Fan_Start := FALSE
    Physical_Blocked        : BOOL;             // Physical needs OFF→ON cycle
    
    Cycle_Count             : UDINT;
    Status_Message          : STRING(50);
END_VAR

VAR
    State                   : UINT;
    Pressurize_Timer        : TON;
    Cooldown_Timer          : TON;
    Feedback_Timer          : TON;
    Post_Dump_Timer         : TON;
    
    Start_Prev              : BOOL;
    Fault_Latched           : BOOL;
    Physical_Was_Off        : BOOL;
    Controlled_Stop_Active  : BOOL;
    Temp_Stop_Active        : BOOL;             // NEW: Temperature dump stop in progress
    Start_Command           : BOOL;
END_VAR

// ============================================
// RESET FAULTS
// ============================================
IF Reset_Fault THEN
    Fault_Latched := FALSE;
    Fan_Fault := FALSE;
    Fault_Motor_Overload := FALSE;
    Fault_Pressure := FALSE;
    Fault_Contactor := FALSE;
    Fault_Emergency := FALSE;
    Controlled_Stop_Active := FALSE;
    Temp_Stop_Active := FALSE;
    Post_Dump_Timer(IN := FALSE);
    Cooldown_Timer(IN := FALSE);
    IF State = 99 THEN
        State := 0;
    END_IF;
END_IF;

// ============================================
// FORCE HMI OFF (when fault or controlled stop)
// ============================================
Force_HMI_Off := Fault_Latched OR Controlled_Stop_Active OR Temp_Stop_Active;

// ============================================
// COMBINE START COMMAND
// ============================================
IF Physical_Enabled THEN
    Start_Command := HMI_Start AND Physical_Start AND NOT Force_HMI_Off;
ELSE
    Start_Command := HMI_Start AND NOT Force_HMI_Off;
END_IF;

// ============================================
// PHYSICAL BUTTON BLOCKING (needs OFF→ON cycle)
// ============================================
IF Fault_Latched AND Physical_Enabled THEN
    Physical_Blocked := TRUE;
    Physical_Was_Off := FALSE;
ELSIF Physical_Blocked THEN
    IF NOT Physical_Start THEN
        Physical_Was_Off := TRUE;
    END_IF;
    
    IF Physical_Was_Off AND NOT Fault_Latched THEN
        Physical_Blocked := FALSE;
        Physical_Was_Off := FALSE;
    END_IF;
END_IF;

// ============================================
// EMERGENCY IMMEDIATE - STOP NOW
// ============================================
IF Emergency_Immediate THEN
    Contactor_Output := FALSE;
    Fan_Running := FALSE;
    Fan_Pressurized := FALSE;
    Fault_Emergency := TRUE;
    Fault_Latched := TRUE;
    Fan_Fault := TRUE;
    Controlled_Stop_Active := FALSE;
    Temp_Stop_Active := FALSE;
    State := 99;
    Status_Message := 'IMMEDIATE E-STOP - FAN OFF';
    RETURN;
END_IF;

// ============================================
// EMERGENCY CONTROLLED - FAN STAYS ON DURING DUMP
// Then stops after Post_Dump_Delay (short)
// ============================================
IF Emergency_Controlled AND NOT Temp_Stop_Active THEN
    Controlled_Stop_Active := TRUE;
    
    IF NOT Dump_Complete THEN
        Status_Message := 'EMG CTRL - DUMPING LOAD';
    ELSE
        // Dump complete - start short delay before fan stop
        Post_Dump_Timer(IN := TRUE, PT := Post_Dump_Delay);
        Status_Message := 'EMG CTRL - FAN STOPPING';
        
        IF Post_Dump_Timer.Q THEN
            Contactor_Output := FALSE;
            Fan_Running := FALSE;
            Fan_Pressurized := FALSE;
            Fault_Emergency := TRUE;
            Fault_Latched := TRUE;
            Fan_Fault := TRUE;
            Controlled_Stop_Active := FALSE;
            Post_Dump_Timer(IN := FALSE);
            State := 99;
            Status_Message := 'EMG COMPLETE - RESET REQ';
            RETURN;
        END_IF;
    END_IF;
END_IF;

// Clear EMG controlled when signal goes away (if not latched)
IF NOT Emergency_Controlled AND NOT Fault_Latched AND Controlled_Stop_Active THEN
    Controlled_Stop_Active := FALSE;
    Post_Dump_Timer(IN := FALSE);
END_IF;

// ============================================
// TEMPERATURE DUMP - FAN STAYS ON DURING DUMP
// Then goes to FULL COOLDOWN (same as normal stop)
// ============================================
IF Is_Temperature_Dump AND NOT Emergency_Controlled AND NOT Controlled_Stop_Active THEN
    Temp_Stop_Active := TRUE;
    
    IF NOT Dump_Complete THEN
        Status_Message := 'OVER TEMP - DUMPING LOAD';
    ELSE
        // Dump complete - go to cooldown state (state 40)
        // Fan keeps running for full cooldown time
        IF State <> 40 AND State <> 99 THEN
            State := 40;
            Cooldown_Timer(IN := FALSE);  // Reset timer to start fresh
            Status_Message := 'TEMP - COOLING DOWN';
        END_IF;
    END_IF;
END_IF;

// ============================================
// MOTOR OVERLOAD CHECK
// ============================================
IF Contactor_Output AND NOT Motor_Overload_OK THEN
    Fault_Motor_Overload := TRUE;
    Fault_Latched := TRUE;
    Fan_Fault := TRUE;
    Contactor_Output := FALSE;
    Fan_Running := FALSE;
    Fan_Pressurized := FALSE;
    Controlled_Stop_Active := FALSE;
    Temp_Stop_Active := FALSE;
    State := 99;
    Status_Message := 'MOTOR OVERLOAD FAULT';
    RETURN;
END_IF;

// ============================================
// FAULT LATCHED - STAY STOPPED
// Exception: Controlled E-Stop or Temp dump keeps fan running
// ============================================
IF Fault_Latched AND NOT Controlled_Stop_Active AND NOT Temp_Stop_Active THEN
    Contactor_Output := FALSE;
    Fan_Running := FALSE;
    Fan_Pressurized := FALSE;
    Status_Message := 'FAULT - RESET REQUIRED';
    RETURN;
END_IF;

// Physical blocked check
IF Physical_Enabled AND Physical_Blocked THEN
    Contactor_Output := FALSE;
    Fan_Running := FALSE;
    Fan_Pressurized := FALSE;
    Status_Message := 'CYCLE PHYSICAL OFF-ON';
    RETURN;
END_IF;

// ============================================
// NOT ENABLED
// ============================================
IF NOT Enable AND NOT Controlled_Stop_Active AND NOT Temp_Stop_Active THEN
    Contactor_Output := FALSE;
    Fan_Running := FALSE;
    Fan_Pressurized := FALSE;
    State := 0;
    Status_Message := 'FAN OFF';
    Pressurize_Timer(IN := FALSE);
    Cooldown_Timer(IN := FALSE);
    Feedback_Timer(IN := FALSE);
    RETURN;
END_IF;

// ============================================
// STATE MACHINE
// ============================================
CASE State OF

    0: // OFF
        Contactor_Output := FALSE;
        Fan_Running := FALSE;
        Fan_Pressurized := FALSE;
        Status_Message := 'FAN OFF';
        
        Pressurize_Timer(IN := FALSE);
        Cooldown_Timer(IN := FALSE);
        Feedback_Timer(IN := FALSE);
        
        IF Start_Command AND NOT Start_Prev THEN
            State := 10;
            Cycle_Count := Cycle_Count + 1;
        END_IF;
    
    10: // STARTING
        Contactor_Output := TRUE;
        Fan_Running := FALSE;
        Fan_Pressurized := FALSE;
        Status_Message := 'FAN STARTING';
        
        Feedback_Timer(IN := NOT Contactor_Feedback, PT := Feedback_Timeout);
        
        IF Feedback_Timer.Q THEN
            Fault_Contactor := TRUE;
            Fault_Latched := TRUE;
            Fan_Fault := TRUE;
            Status_Message := 'CONTACTOR FAULT';
            State := 99;
        ELSIF Contactor_Feedback THEN
            Feedback_Timer(IN := FALSE);
            State := 20;
        END_IF;
    
    20: // PRESSURIZING
        Contactor_Output := TRUE;
        Fan_Running := FALSE;
        Fan_Pressurized := FALSE;
        Status_Message := 'FAN PRESSURIZING';
        
        Pressurize_Timer(IN := TRUE, PT := Pressurize_Time);
        
        IF Pressurize_Timer.Q THEN
            IF Pressure_OK THEN
                Fan_Pressurized := TRUE;
                Pressurize_Timer(IN := FALSE);
                State := 30;
            ELSE
                Fault_Pressure := TRUE;
                Fault_Latched := TRUE;
                Fan_Fault := TRUE;
                Status_Message := 'PRESSURE FAULT';
                State := 99;
            END_IF;
        END_IF;
        
        IF NOT Start_Command AND NOT Controlled_Stop_Active AND NOT Temp_Stop_Active THEN
            Pressurize_Timer(IN := FALSE);
            State := 40;
        END_IF;
    
    30: // RUNNING
        Contactor_Output := TRUE;
        Fan_Running := TRUE;
        Fan_Pressurized := TRUE;
        
        // Don't overwrite status if in controlled/temp stop
        IF NOT Controlled_Stop_Active AND NOT Temp_Stop_Active THEN
            Status_Message := 'FAN RUNNING';
        END_IF;
        
        IF NOT Pressure_OK THEN
            Fault_Pressure := TRUE;
            Fault_Latched := TRUE;
            Fan_Fault := TRUE;
            Controlled_Stop_Active := FALSE;
            Temp_Stop_Active := FALSE;
            Status_Message := 'PRESSURE LOSS FAULT';
            State := 99;
        END_IF;
        
        IF NOT Start_Command AND NOT Controlled_Stop_Active AND NOT Temp_Stop_Active THEN
            State := 40;
        END_IF;
    
    40: // COOLING DOWN (used for normal stop AND temperature dump)
        Contactor_Output := TRUE;
        Fan_Running := FALSE;
        Fan_Pressurized := FALSE;
        
        Cooldown_Timer(IN := TRUE, PT := Cooldown_Time);
        
        // Calculate remaining time for display
        IF Temp_Stop_Active THEN
            Status_Message := 'TEMP COOLDOWN';
        ELSE
            Status_Message := 'FAN COOLING DOWN';
        END_IF;
        
        IF Cooldown_Timer.Q THEN
            Cooldown_Timer(IN := FALSE);
            Contactor_Output := FALSE;
            
            // If this was temp stop, set fault to require reset
            IF Temp_Stop_Active THEN
                Fault_Emergency := TRUE;
                Fault_Latched := TRUE;
                Fan_Fault := TRUE;
                Temp_Stop_Active := FALSE;
                Status_Message := 'TEMP STOP COMPLETE';
                State := 99;
            ELSE
                Status_Message := 'FAN OFF';
                State := 0;
            END_IF;
        END_IF;
    
    99: // FAULT
        Contactor_Output := FALSE;
        Fan_Running := FALSE;
        Fan_Pressurized := FALSE;
        Fan_Fault := TRUE;

END_CASE;

Start_Prev := Start_Command;

END_FUNCTION_BLOCK

// ---- POUs/FB_Temperature_Monitor.TcPOU
FUNCTION_BLOCK FB_Temperature_Monitor
VAR_INPUT
    // TC Readings
    Outlet_TC_Readings      : ARRAY[1..4] OF REAL;
    Inlet_TC_Reading        : REAL;
    
    // Configuration
    Outlet_TC_Count         : UINT := 2;                // 2 or 4 only
    Inlet_TC_Enabled        : BOOL := TRUE;
    
    // Outlet TC Thresholds
    Outlet_Warning_Temp     : REAL := 350.0;
    Outlet_Maximum_Temp     : REAL := 400.0;
    TC_Open_Limit           : REAL := 700.0;            // Above = TC open
    TC_Short_Limit          : REAL := -50.0;            // Below = TC shorted
    
    // Inlet TC Thresholds
    Inlet_Warning_Temp      : REAL := 50.0;
    Inlet_Maximum_Temp      : REAL := 75.0;
    
    Enable                  : BOOL;
    Reset                   : BOOL;
END_VAR

VAR_OUTPUT
    // Calculated values
    Outlet_Temp_Avg         : REAL;
    Outlet_Temp_Max         : REAL;
    Inlet_Temp              : REAL;
    Delta_T                 : REAL;
    Hottest_TC_Index        : UINT;
    
    // Individual OUTLET TC Fail (for alarm page)
    Outlet_TC1_Fail         : BOOL;
    Outlet_TC2_Fail         : BOOL;
    Outlet_TC3_Fail         : BOOL;
    Outlet_TC4_Fail         : BOOL;
    
    // Individual OUTLET TC Warning (for alarm page)
    Outlet_TC1_Warning      : BOOL;
    Outlet_TC2_Warning      : BOOL;
    Outlet_TC3_Warning      : BOOL;
    Outlet_TC4_Warning      : BOOL;
    
    // Individual OUTLET TC Overtemp (for alarm page)
    Outlet_TC1_Overtemp     : BOOL;
    Outlet_TC2_Overtemp     : BOOL;
    Outlet_TC3_Overtemp     : BOOL;
    Outlet_TC4_Overtemp     : BOOL;
    
    // INLET TC Status (for alarm page)
    Inlet_TC_Fail           : BOOL;
    Inlet_TC_Warning        : BOOL;
    Inlet_TC_Overtemp       : BOOL;
    
    // Combined status
    TC_Fail_Dump_Required   : BOOL;                     // TC fail requires dump
    Any_Warning             : BOOL;
    Any_Overtemp            : BOOL;
    Contingency_Mode        : BOOL;                     // Running with backup TC (4 TC only)
    
    Dump_Command            : BOOL;
    
    Status_Text             : STRING(100);
END_VAR

VAR
    i                       : UINT;
    TempSum                 : REAL;
    ValidCount              : UINT;
    
    TC_Fail_Arr             : ARRAY[1..4] OF BOOL;
    TC_Warning_Arr          : ARRAY[1..4] OF BOOL;
    TC_Overtemp_Arr         : ARRAY[1..4] OF BOOL;
    TC_Valid_Arr            : ARRAY[1..4] OF BOOL;
    
    Warning_Latched         : BOOL;
    Overtemp_Latched        : BOOL;
    
    Side1_Failed            : BOOL;                     // TC1 + TC2 both failed
    Side2_Failed            : BOOL;                     // TC3 + TC4 both failed
END_VAR

// ============================================
// RESET
// ============================================
IF Reset THEN
    Outlet_TC1_Fail := FALSE;
    Outlet_TC2_Fail := FALSE;
    Outlet_TC3_Fail := FALSE;
    Outlet_TC4_Fail := FALSE;
    
    Outlet_TC1_Warning := FALSE;
    Outlet_TC2_Warning := FALSE;
    Outlet_TC3_Warning := FALSE;
    Outlet_TC4_Warning := FALSE;
    
    Outlet_TC1_Overtemp := FALSE;
    Outlet_TC2_Overtemp := FALSE;
    Outlet_TC3_Overtemp := FALSE;
    Outlet_TC4_Overtemp := FALSE;
    
    Inlet_TC_Fail := FALSE;
    Inlet_TC_Warning := FALSE;
    Inlet_TC_Overtemp := FALSE;
    
    TC_Fail_Dump_Required := FALSE;
    Warning_Latched := FALSE;
    Overtemp_Latched := FALSE;
    Contingency_Mode := FALSE;
END_IF;

// ============================================
// NOT ENABLED
// ============================================
IF NOT Enable THEN
    Any_Warning := FALSE;
    Any_Overtemp := FALSE;
    Dump_Command := FALSE;
    Status_Text := 'Temp monitoring disabled';
    RETURN;
END_IF;

// ============================================
// CHECK EACH OUTLET TC - HEALTH AND TEMPERATURE
// ============================================
FOR i := 1 TO 4 DO
    TC_Fail_Arr[i] := FALSE;
    TC_Warning_Arr[i] := FALSE;
    TC_Overtemp_Arr[i] := FALSE;
    TC_Valid_Arr[i] := FALSE;
    
    IF i <= Outlet_TC_Count THEN
        // TC Health Check
        IF Outlet_TC_Readings[i] > TC_Open_Limit OR Outlet_TC_Readings[i] < TC_Short_Limit THEN
            TC_Fail_Arr[i] := TRUE;
        ELSE
            TC_Valid_Arr[i] := TRUE;
            
            // Temperature Check
            IF Outlet_TC_Readings[i] >= Outlet_Maximum_Temp THEN
                TC_Overtemp_Arr[i] := TRUE;
            ELSIF Outlet_TC_Readings[i] >= Outlet_Warning_Temp THEN
                TC_Warning_Arr[i] := TRUE;
            END_IF;
        END_IF;
    END_IF;
END_FOR;

// Copy to individual outputs (for alarm page)
Outlet_TC1_Fail := TC_Fail_Arr[1];
Outlet_TC2_Fail := TC_Fail_Arr[2];
Outlet_TC3_Fail := TC_Fail_Arr[3];
Outlet_TC4_Fail := TC_Fail_Arr[4];

Outlet_TC1_Warning := TC_Warning_Arr[1];
Outlet_TC2_Warning := TC_Warning_Arr[2];
Outlet_TC3_Warning := TC_Warning_Arr[3];
Outlet_TC4_Warning := TC_Warning_Arr[4];

Outlet_TC1_Overtemp := TC_Overtemp_Arr[1];
Outlet_TC2_Overtemp := TC_Overtemp_Arr[2];
Outlet_TC3_Overtemp := TC_Overtemp_Arr[3];
Outlet_TC4_Overtemp := TC_Overtemp_Arr[4];

// ============================================
// CHECK INLET TC (if enabled)
// ============================================
IF Inlet_TC_Enabled THEN
    IF Inlet_TC_Reading > TC_Open_Limit OR Inlet_TC_Reading < TC_Short_Limit THEN
        Inlet_TC_Fail := TRUE;
        Inlet_TC_Warning := FALSE;
        Inlet_TC_Overtemp := FALSE;
    ELSE
        Inlet_TC_Fail := FALSE;
        
        IF Inlet_TC_Reading >= Inlet_Maximum_Temp THEN
            Inlet_TC_Overtemp := TRUE;
            Inlet_TC_Warning := FALSE;
        ELSIF Inlet_TC_Reading >= Inlet_Warning_Temp THEN
            Inlet_TC_Warning := TRUE;
            Inlet_TC_Overtemp := FALSE;
        ELSE
            Inlet_TC_Warning := FALSE;
            Inlet_TC_Overtemp := FALSE;
        END_IF;
    END_IF;
ELSE
    Inlet_TC_Fail := FALSE;
    Inlet_TC_Warning := FALSE;
    Inlet_TC_Overtemp := FALSE;
END_IF;

// ============================================
// TC FAIL LOGIC
// 2 TCs: ANY fail = DUMP
// 4 TCs: Both same side fail = DUMP
// ============================================
Side1_Failed := FALSE;
Side2_Failed := FALSE;
TC_Fail_Dump_Required := FALSE;
Contingency_Mode := FALSE;

CASE Outlet_TC_Count OF
    2:
        // 2 TCs: ANY single fail = DUMP (no backup)
        IF TC_Fail_Arr[1] OR TC_Fail_Arr[2] THEN
            TC_Fail_Dump_Required := TRUE;
        END_IF;
        
    4:
        // Check Side 1 (TC1 + TC2)
        IF TC_Fail_Arr[1] AND TC_Fail_Arr[2] THEN
            Side1_Failed := TRUE;
            TC_Fail_Dump_Required := TRUE;
        END_IF;
        
        // Check Side 2 (TC3 + TC4)
        IF TC_Fail_Arr[3] AND TC_Fail_Arr[4] THEN
            Side2_Failed := TRUE;
            TC_Fail_Dump_Required := TRUE;
        END_IF;
        
        // Contingency = any single fail but not both on same side
        IF (TC_Fail_Arr[1] OR TC_Fail_Arr[2] OR TC_Fail_Arr[3] OR TC_Fail_Arr[4]) 
           AND NOT TC_Fail_Dump_Required THEN
            Contingency_Mode := TRUE;
        END_IF;
        
    ELSE
        TC_Fail_Dump_Required := TRUE;
        Status_Text := 'Invalid TC count (2 or 4)';
END_CASE;

// ============================================
// CALCULATE AVERAGE AND FIND MAX (valid TCs only)
// ============================================
TempSum := 0.0;
ValidCount := 0;
Outlet_Temp_Max := -999.0;
Hottest_TC_Index := 0;

FOR i := 1 TO Outlet_TC_Count DO
    IF TC_Valid_Arr[i] THEN
        TempSum := TempSum + Outlet_TC_Readings[i];
        ValidCount := ValidCount + 1;
        
        IF Outlet_TC_Readings[i] > Outlet_Temp_Max THEN
            Outlet_Temp_Max := Outlet_TC_Readings[i];
            Hottest_TC_Index := i;
        END_IF;
    END_IF;
END_FOR;

IF ValidCount > 0 THEN
    Outlet_Temp_Avg := TempSum / UINT_TO_REAL(ValidCount);
ELSE
    Outlet_Temp_Avg := 0.0;
    Outlet_Temp_Max := 0.0;
END_IF;

// Store inlet value
IF Inlet_TC_Enabled AND NOT Inlet_TC_Fail THEN
    Inlet_Temp := Inlet_TC_Reading;
    Delta_T := Outlet_Temp_Max - Inlet_Temp;
ELSE
    Inlet_Temp := 0.0;
    Delta_T := 0.0;
END_IF;

// ============================================
// COMBINED STATUS
// ============================================
Any_Warning := TC_Warning_Arr[1] OR TC_Warning_Arr[2] OR TC_Warning_Arr[3] OR TC_Warning_Arr[4] OR Inlet_TC_Warning;
Any_Overtemp := TC_Overtemp_Arr[1] OR TC_Overtemp_Arr[2] OR TC_Overtemp_Arr[3] OR TC_Overtemp_Arr[4] OR Inlet_TC_Overtemp;

// Latch alarms
IF Any_Warning THEN
    Warning_Latched := TRUE;
END_IF;

IF Any_Overtemp THEN
    Overtemp_Latched := TRUE;
END_IF;

// ============================================
// DUMP COMMAND
// ============================================
Dump_Command := Any_Overtemp OR TC_Fail_Dump_Required OR (Inlet_TC_Enabled AND Inlet_TC_Fail);

// ============================================
// STATUS MESSAGE
// ============================================
IF Outlet_TC_Count = 2 THEN
    IF TC_Fail_Arr[1] AND TC_Fail_Arr[2] THEN
        Status_Text := 'TC1+TC2 FAIL - DUMPING';
    ELSIF TC_Fail_Arr[1] THEN
        Status_Text := 'TC1 FAIL - DUMPING';
    ELSIF TC_Fail_Arr[2] THEN
        Status_Text := 'TC2 FAIL - DUMPING';
    END_IF;
ELSIF Outlet_TC_Count = 4 THEN
    IF Side1_Failed AND Side2_Failed THEN
        Status_Text := 'ALL TCs FAIL - DUMPING';
    ELSIF Side1_Failed THEN
        Status_Text := 'TC1+TC2 FAIL - DUMPING';
    ELSIF Side2_Failed THEN
        Status_Text := 'TC3+TC4 FAIL - DUMPING';
    END_IF;
END_IF;

// Override with other conditions
IF Inlet_TC_Enabled AND Inlet_TC_Fail THEN
    Status_Text := 'INLET TC FAIL - DUMPING';
ELSIF Inlet_TC_Overtemp THEN
    Status_Text := 'INLET OVERTEMP - DUMPING';
ELSIF Any_Overtemp THEN
    Status_Text := 'OUTLET OVERTEMP - DUMPING';
ELSIF Contingency_Mode THEN
    Status_Text := 'CONTINGENCY MODE';
ELSIF Inlet_TC_Warning THEN
    Status_Text := 'INLET TEMP WARNING';
ELSIF Any_Warning THEN
    Status_Text := 'OUTLET TEMP WARNING';
ELSIF Warning_Latched OR Overtemp_Latched THEN
    Status_Text := 'Alarm history - reset';
ELSIF NOT TC_Fail_Dump_Required THEN
    Status_Text := 'Normal';
END_IF;

END_FUNCTION_BLOCK

// ---- POUs/FB_Gradual_Dump.TcPOU
FUNCTION_BLOCK FB_Gradual_Dump
// ============================================
// GRADUAL DUMP CONTROLLER
// UPDATED: Separate settings for EMG vs TEMP dump
// - EMG dump: Uses LB_EMG_DUMP_PERCENT / LB_EMG_DUMP_STEP_TIME
// - TEMP dump: Uses LB_TEMP_DUMP_PERCENT / LB_TEMP_DUMP_STEP_TIME
// ============================================

VAR_INPUT
    // Separate triggers (to know which type)
    Temp_Dump_Trigger       : BOOL;             // From Temp Monitor
    EMG_Dump_Trigger        : BOOL;             // From E-Stop Controlled
    
    // Current load info
    Current_Power_kW        : REAL;
    Rated_Power_kW          : REAL;
    
    // EMG dump configuration (from ENG page)
    EMG_Percent_Per_Step    : REAL := 10.0;     // NEW: % per step for EMG
    EMG_Step_Time           : TIME := T#1s;     // NEW: Time between steps for EMG
    
    // TEMP dump configuration (from ENG page)
    Temp_Percent_Per_Step   : REAL := 10.0;     // NEW: % per step for temp
    Temp_Step_Time          : TIME := T#2s;     // NEW: Time between steps for temp
    
    // Safety timeout
    Dump_Timeout            : TIME := T#30s;
    
    Enable                  : BOOL;
    Reset                   : BOOL;
END_VAR

VAR_OUTPUT
    Dump_Active             : BOOL;
    Dump_Complete           : BOOL;
    Dump_Percent            : REAL := 100.0;    // Current % remaining (100 → 0)
    Dump_Timeout_Fault      : BOOL;
    
    // Type of dump (for fan control)
    Is_Temperature_Dump     : BOOL;             // Fan uses full cooldown
    Is_Emergency_Dump       : BOOL;             // Fan uses short delay
    
    Target_Power_kW         : REAL;
    
    Status_Text             : STRING(100);
END_VAR

VAR
    State                   : UINT;
    Step_Timer              : TON;
    Timeout_Timer           : TON;
    
    Initial_Power_kW        : REAL;
    Temp_Dump_Latched       : BOOL;
    EMG_Dump_Latched        : BOOL;
    
    // Active settings based on dump type
    Active_Percent          : REAL;             // NEW: Which percent to use
    Active_Step_Time        : TIME;             // NEW: Which time to use
END_VAR

// ============================================
// RESET
// ============================================
IF Reset THEN
    Dump_Active := FALSE;
    Dump_Complete := FALSE;
    Dump_Percent := 100.0;
    Dump_Timeout_Fault := FALSE;
    Is_Temperature_Dump := FALSE;
    Is_Emergency_Dump := FALSE;
    Temp_Dump_Latched := FALSE;
    EMG_Dump_Latched := FALSE;
    State := 0;
    Step_Timer(IN := FALSE);
    Timeout_Timer(IN := FALSE);
    Status_Text := 'Reset';
END_IF;

// ============================================
// NOT ENABLED
// ============================================
IF NOT Enable THEN
    Dump_Active := FALSE;
    Dump_Percent := 100.0;
    Target_Power_kW := Rated_Power_kW;
    Status_Text := 'Disabled';
    RETURN;
END_IF;

// ============================================
// LATCH DUMP TRIGGERS
// Once triggered, dump continues until complete
// EMG takes priority if both trigger
// ============================================
IF Temp_Dump_Trigger AND NOT Dump_Complete AND NOT EMG_Dump_Latched THEN
    Temp_Dump_Latched := TRUE;
END_IF;

IF EMG_Dump_Trigger AND NOT Dump_Complete THEN
    EMG_Dump_Latched := TRUE;
    Temp_Dump_Latched := FALSE;  // EMG overrides temp
END_IF;

// Set dump type outputs
Is_Temperature_Dump := Temp_Dump_Latched AND NOT EMG_Dump_Latched;
Is_Emergency_Dump := EMG_Dump_Latched;

// ============================================
// SELECT ACTIVE DUMP RATE BASED ON TYPE
// ============================================
IF EMG_Dump_Latched THEN
    Active_Percent := EMG_Percent_Per_Step;
    Active_Step_Time := EMG_Step_Time;
ELSE
    Active_Percent := Temp_Percent_Per_Step;
    Active_Step_Time := Temp_Step_Time;
END_IF;

// ============================================
// STATE MACHINE
// ============================================
CASE State OF

    0: // IDLE - Waiting for dump trigger
        Dump_Active := FALSE;
        Dump_Complete := FALSE;
        Dump_Percent := 100.0;
        Target_Power_kW := Rated_Power_kW;
        Status_Text := 'Ready';
        
        Step_Timer(IN := FALSE);
        Timeout_Timer(IN := FALSE);
        
        IF Temp_Dump_Latched OR EMG_Dump_Latched THEN
            Initial_Power_kW := Current_Power_kW;
            Dump_Active := TRUE;
            State := 10;
            
            // Set initial status message
            IF EMG_Dump_Latched THEN
                Status_Text := 'CONTROLLED E-STOP - STARTING DUMP';
            ELSE
                Status_Text := 'OVER TEMPERATURE - STARTING DUMP';
            END_IF;
        END_IF;
    
    10: // DUMPING - Gradually reduce load
        Dump_Active := TRUE;
        Dump_Complete := FALSE;
        
        // Status message with progress
        IF Is_Emergency_Dump THEN
            Status_Text := CONCAT('EMG DUMPING - ', REAL_TO_STRING(Dump_Percent));
            Status_Text := CONCAT(Status_Text, '% remaining');
        ELSE
            Status_Text := CONCAT('TEMP DUMPING - ', REAL_TO_STRING(Dump_Percent));
            Status_Text := CONCAT(Status_Text, '% remaining');
        END_IF;
        
        // Timeout protection
        Timeout_Timer(IN := TRUE, PT := Dump_Timeout);
        IF Timeout_Timer.Q THEN
            Dump_Timeout_Fault := TRUE;
            Dump_Percent := 0.0;
            Status_Text := 'DUMP TIMEOUT - FORCED TO 0%';
            State := 20;
        END_IF;
        
        // Step timer - uses ACTIVE settings based on dump type
        Step_Timer(IN := TRUE, PT := Active_Step_Time);
        
        IF Step_Timer.Q THEN
            Dump_Percent := Dump_Percent - Active_Percent;
            
            IF Dump_Percent <= 0.0 THEN
                Dump_Percent := 0.0;
                State := 20;
            END_IF;
            
            Step_Timer(IN := FALSE);
        END_IF;
        
        Target_Power_kW := (Dump_Percent / 100.0) * Rated_Power_kW;
    
    20: // COMPLETE - Dump finished
        Dump_Active := FALSE;
        Dump_Complete := TRUE;
        Dump_Percent := 0.0;
        Target_Power_kW := 0.0;
        
        IF Dump_Timeout_Fault THEN
            Status_Text := 'DUMP TIMEOUT - ALL LOADS OFF';
        ELSIF Is_Emergency_Dump THEN
            Status_Text := 'EMG DUMP COMPLETE - ALL LOADS OFF';
        ELSE
            Status_Text := 'TEMP DUMP COMPLETE - COOLING DOWN';
        END_IF;
        
        Step_Timer(IN := FALSE);
        Timeout_Timer(IN := FALSE);

END_CASE;

END_FUNCTION_BLOCK

// ---- POUs/FB_Main_Contactor.TcPOU
FUNCTION_BLOCK FB_Main_Contactor
VAR_INPUT
    // Enable conditions
    Master_Enable           : BOOL;
    Fan_Running             : BOOL;
    Fan_Pressurized         : BOOL;
    
    // Block conditions
    Any_Alarm               : BOOL;
    Dump_Active             : BOOL;
    Dump_Complete           : BOOL;
    Is_Temperature_Dump     : BOOL;             // TRUE = fan stays on, can recover
    
    // Feedback
    Contactor_Feedback      : BOOL;             // NO contact: TRUE = closed
    
    // Configuration
    Feedback_Timeout        : TIME := T#3s;
    
    Enable                  : BOOL;
    Reset                   : BOOL;
END_VAR

VAR_OUTPUT
    Contactor_Output        : BOOL;
    Contactor_Closed        : BOOL;             // Confirmed closed
    
    Contactor_Fault         : BOOL;
    Fault_No_Feedback       : BOOL;             // Commanded ON but no feedback
    Fault_Stuck_Closed      : BOOL;             // Commanded OFF but still closed
    
    Status_Text             : STRING(50);
END_VAR

VAR
    Feedback_Timer          : TON;
    Stuck_Timer             : TON;
    
    Fault_Latched           : BOOL;
    Contactor_Allowed       : BOOL;
END_VAR

// ============================================
// RESET
// ============================================
IF Reset THEN
    Fault_Latched := FALSE;
    Contactor_Fault := FALSE;
    Fault_No_Feedback := FALSE;
    Fault_Stuck_Closed := FALSE;
    Feedback_Timer(IN := FALSE);
    Stuck_Timer(IN := FALSE);
END_IF;

// ============================================
// NOT ENABLED
// ============================================
IF NOT Enable THEN
    Contactor_Output := FALSE;
    Contactor_Closed := FALSE;
    Status_Text := 'Disabled';
    RETURN;
END_IF;

// ============================================
// FAULT LATCHED
// ============================================
IF Fault_Latched THEN
    Contactor_Output := FALSE;
    Contactor_Closed := FALSE;
    Status_Text := 'FAULT - Reset required';
    RETURN;
END_IF;

// ============================================
// CONTACTOR ALLOWED LOGIC
// ============================================
Contactor_Allowed := 
    Master_Enable
    AND Fan_Running
    AND Fan_Pressurized
    AND NOT Any_Alarm
    AND NOT Dump_Active
    AND NOT Dump_Complete;

// Special case: Temperature dump recovery
// After reset, dump flags clear, contactor allowed again

// ============================================
// CONTACTOR OUTPUT
// ============================================
IF Contactor_Allowed THEN
    Contactor_Output := TRUE;
ELSE
    Contactor_Output := FALSE;
END_IF;

// ============================================
// FEEDBACK MONITORING - NO FEEDBACK
// Commanded ON but no feedback within timeout
// ============================================
Feedback_Timer(IN := Contactor_Output AND NOT Contactor_Feedback, PT := Feedback_Timeout);

IF Feedback_Timer.Q THEN
    Fault_No_Feedback := TRUE;
    Fault_Latched := TRUE;
    Contactor_Fault := TRUE;
    Contactor_Output := FALSE;
    Status_Text := 'FAULT - No feedback';
    RETURN;
END_IF;

// ============================================
// FEEDBACK MONITORING - STUCK CLOSED
// Commanded OFF but feedback still TRUE
// ============================================
Stuck_Timer(IN := NOT Contactor_Output AND Contactor_Feedback, PT := Feedback_Timeout);

IF Stuck_Timer.Q THEN
    Fault_Stuck_Closed := TRUE;
    Fault_Latched := TRUE;
    Contactor_Fault := TRUE;
    Status_Text := 'FAULT - Stuck closed';
    RETURN;
END_IF;

// ============================================
// CONTACTOR STATUS
// ============================================
Contactor_Closed := Contactor_Output AND Contactor_Feedback;

// ============================================
// STATUS MESSAGE
// ============================================
IF Contactor_Closed THEN
    Status_Text := 'Closed';
ELSIF Contactor_Output AND NOT Contactor_Feedback THEN
    Status_Text := 'Closing...';
ELSIF NOT Contactor_Output AND Contactor_Feedback THEN
    Status_Text := 'Opening...';
ELSIF NOT Master_Enable THEN
    Status_Text := 'No Master Enable';
ELSIF NOT Fan_Running THEN
    Status_Text := 'Fan not running';
ELSIF NOT Fan_Pressurized THEN
    Status_Text := 'Not pressurized';
ELSIF Any_Alarm THEN
    Status_Text := 'Alarm active';
ELSIF Dump_Active THEN
    Status_Text := 'Dump active';
ELSIF Dump_Complete THEN
    Status_Text := 'Dump complete';
ELSE
    Status_Text := 'Open';
END_IF;

END_FUNCTION_BLOCK

// ---- POUs/FB_Load_Controller.TcPOU
FUNCTION_BLOCK FB_Load_Controller
// ============================================
// LOAD CONTROLLER
// - Power grouping (steps grouped by kW rating)
// - Step feedback monitoring
// - Total power monitoring
// - Step quarantine management
// - Wear leveling by cycle count
// ============================================

VAR_INPUT
    // Target from mode or dump
    Target_Power_kW         : REAL;
    
    // Main contactor status
    Main_Contactor_Closed   : BOOL;
    
    // Step configuration
    Step_Power_Rating       : ARRAY[1..LB_NUMBER_OF_STEPS] OF REAL;
    Number_Of_Steps         : UINT := 10;
    
    // Step feedback from IO
    Step_Feedback           : ARRAY[1..LB_NUMBER_OF_STEPS] OF BOOL;
    
    // Total power from power meter
    Measured_Total_Power    : REAL;
    
    // Manual quarantine from HMI
    Step_Quarantine_Manual  : ARRAY[1..LB_NUMBER_OF_STEPS] OF BOOL;
    Step_Unquarantine_Cmd   : ARRAY[1..LB_NUMBER_OF_STEPS] OF BOOL;
    
    // Maintenance mode
    Maintenance_Mode        : BOOL;
    Manual_Step_Cmd         : ARRAY[1..LB_NUMBER_OF_STEPS] OF BOOL;
    
    // Configuration (from ENG page)
    Deadband_kW             : REAL := 5.0;
    Step_Up_Delay           : TIME := T#500ms;
    Step_Down_Delay         : TIME := T#500ms;
    Feedback_Timeout        : TIME := T#3s;
    Enable_Feedback_Monitoring : BOOL := TRUE;
    
    // Total power monitoring config
    Power_Tolerance_Percent : REAL := 5.0;
    Power_Monitor_Delay     : TIME := T#10s;
    Enable_Power_Monitoring : BOOL := TRUE;
    
    Enable                  : BOOL;
    Reset                   : BOOL;
END_VAR

VAR_OUTPUT
    // Coil outputs
    Step_Coil_Cmd           : ARRAY[1..LB_NUMBER_OF_STEPS] OF BOOL;
    
    // Power calculations
    Released_Power_kW       : REAL;
    Available_Power_kW      : REAL;
    Rated_Total_kW          : REAL;
    Power_Error_kW          : REAL;
    At_Target               : BOOL;
    
    // Step counts
    Active_Step_Count       : UINT;
    Quarantined_Step_Count  : UINT;
    Available_Step_Count    : UINT;
    
    // Quarantine status (combined)
    Step_Quarantined        : ARRAY[1..LB_NUMBER_OF_STEPS] OF BOOL;
    Step_Quarantine_Feedback: ARRAY[1..LB_NUMBER_OF_STEPS] OF BOOL;
    
    // Faults
    Any_Feedback_Fault      : BOOL;
    Total_Power_Warning     : BOOL;
    Power_Mismatch_Percent  : REAL;
    
    // Cycle counts (for wear leveling)
    Step_Cycle_Count        : ARRAY[1..LB_NUMBER_OF_STEPS] OF UDINT;
    
    Status_Text             : STRING(100);
END_VAR

VAR
    i                       : UINT;
    j                       : UINT;
    g                       : UINT;
    
    // Internal coil states
    Coil_Internal           : ARRAY[1..LB_NUMBER_OF_STEPS] OF BOOL;
    Coil_Prev               : ARRAY[1..LB_NUMBER_OF_STEPS] OF BOOL;
    
    // Feedback monitoring
    FB_Timer                : ARRAY[1..LB_NUMBER_OF_STEPS] OF TON;
    FB_Fault_Latched        : ARRAY[1..LB_NUMBER_OF_STEPS] OF BOOL;
    
    // Total power monitoring
    Power_Monitor_Timer     : TON;
    Power_Diff              : REAL;
    Expected_Power          : REAL;
    
    // Step change timing
    Step_Up_Timer           : TON;
    Step_Down_Timer         : TON;
    
    // Power grouping - store unique power values (max 20 different sizes)
    Unique_Powers           : ARRAY[1..10] OF REAL;
    Num_Unique_Powers       : UINT;
    Power_Exists            : BOOL;
    Temp_Power              : REAL;
    
    // Distribution calculation
    Current_Power           : REAL;
    Power_Needed            : REAL;
    Best_Step               : UINT;
    Min_Cycles              : UDINT;
    Max_Cycles              : UDINT;
    Step_Available          : BOOL;
    Target_Power_Value      : REAL;
    
    First_Scan              : BOOL := TRUE;
END_VAR

// ============================================
// RESET
// ============================================
IF Reset THEN
    FOR i := 1 TO LB_NUMBER_OF_STEPS DO
        FB_Fault_Latched[i] := FALSE;
        Step_Quarantine_Feedback[i] := FALSE;
    END_FOR;
    Any_Feedback_Fault := FALSE;
    Total_Power_Warning := FALSE;
    Power_Monitor_Timer(IN := FALSE);
END_IF;

// ============================================
// FIRST SCAN - INITIALIZE
// ============================================
IF First_Scan THEN
    FOR i := 1 TO LB_NUMBER_OF_STEPS DO
        Coil_Internal[i] := FALSE;
        Coil_Prev[i] := FALSE;
        FB_Fault_Latched[i] := FALSE;
        Step_Cycle_Count[i] := 0;
    END_FOR;
    First_Scan := FALSE;
END_IF;

// ============================================
// BUILD UNIQUE POWER LIST (sorted largest first)
// ============================================
FOR i := 1 TO 10 DO
    Unique_Powers[i] := 0.0;
END_FOR;
Num_Unique_Powers := 0;

FOR i := 1 TO Number_Of_Steps DO
    IF Step_Power_Rating[i] > 0.0 THEN
        Power_Exists := FALSE;
        
        // Check if this power already in list
        FOR j := 1 TO Num_Unique_Powers DO
            IF Unique_Powers[j] = Step_Power_Rating[i] THEN
                Power_Exists := TRUE;
                EXIT;
            END_IF;
        END_FOR;
        
        // Add new unique power
        IF NOT Power_Exists AND Num_Unique_Powers < 10 THEN
            Num_Unique_Powers := Num_Unique_Powers + 1;
            Unique_Powers[Num_Unique_Powers] := Step_Power_Rating[i];
        END_IF;
    END_IF;
END_FOR;

// Sort unique powers (largest first) - bubble sort
FOR i := 1 TO Num_Unique_Powers - 1 DO
    FOR j := i + 1 TO Num_Unique_Powers DO
        IF Unique_Powers[j] > Unique_Powers[i] THEN
            Temp_Power := Unique_Powers[i];
            Unique_Powers[i] := Unique_Powers[j];
            Unique_Powers[j] := Temp_Power;
        END_IF;
    END_FOR;
END_FOR;

// ============================================
// CALCULATE RATED TOTAL POWER
// ============================================
Rated_Total_kW := 0.0;
FOR i := 1 TO Number_Of_Steps DO
    Rated_Total_kW := Rated_Total_kW + Step_Power_Rating[i];
END_FOR;

// ============================================
// COMBINE QUARANTINE SOURCES
// ============================================
Quarantined_Step_Count := 0;
FOR i := 1 TO Number_Of_Steps DO
    Step_Quarantined[i] := Step_Quarantine_Manual[i] OR Step_Quarantine_Feedback[i];
    
    // Unquarantine command clears feedback quarantine
    IF Step_Unquarantine_Cmd[i] THEN
        Step_Quarantine_Feedback[i] := FALSE;
        FB_Fault_Latched[i] := FALSE;
    END_IF;
    
    IF Step_Quarantined[i] THEN
        Quarantined_Step_Count := Quarantined_Step_Count + 1;
    END_IF;
END_FOR;

// ============================================
// CALCULATE AVAILABLE POWER
// ============================================
Available_Power_kW := 0.0;
Available_Step_Count := 0;
FOR i := 1 TO Number_Of_Steps DO
    IF NOT Step_Quarantined[i] THEN
        Available_Power_kW := Available_Power_kW + Step_Power_Rating[i];
        Available_Step_Count := Available_Step_Count + 1;
    END_IF;
END_FOR;

// ============================================
// NOT ENABLED OR MAIN CONTACTOR OPEN - ALL OFF
// ============================================
IF NOT Enable OR NOT Main_Contactor_Closed THEN
    FOR i := 1 TO LB_NUMBER_OF_STEPS DO
        Coil_Internal[i] := FALSE;
        Step_Coil_Cmd[i] := FALSE;
    END_FOR;
    Released_Power_kW := 0.0;
    Active_Step_Count := 0;
    Power_Error_kW := Target_Power_kW;
    At_Target := (Target_Power_kW <= Deadband_kW);
    
    IF NOT Enable THEN
        Status_Text := 'Disabled';
    ELSE
        Status_Text := 'Main contactor open';
    END_IF;
    RETURN;
END_IF;

// ============================================
// MAINTENANCE MODE - DIRECT CONTROL
// ============================================
IF Maintenance_Mode THEN
    FOR i := 1 TO Number_Of_Steps DO
        Coil_Internal[i] := Manual_Step_Cmd[i] AND NOT Step_Quarantined[i];
    END_FOR;
    Status_Text := 'Maintenance mode';
ELSE

// ============================================
// STEP DISTRIBUTION - POWER GROUP ALGORITHM
// ============================================

// Calculate current released power
Current_Power := 0.0;
Active_Step_Count := 0;
FOR i := 1 TO Number_Of_Steps DO
    IF Coil_Internal[i] THEN
        Current_Power := Current_Power + Step_Power_Rating[i];
        Active_Step_Count := Active_Step_Count + 1;
    END_IF;
END_FOR;

Power_Needed := Target_Power_kW - Current_Power;
Power_Error_kW := Power_Needed;
At_Target := (ABS(Power_Needed) <= Deadband_kW);

// ============================================
// NEED TO ADD POWER?
// ============================================
IF Power_Needed > Deadband_kW THEN
    Step_Up_Timer(IN := TRUE, PT := Step_Up_Delay);
    Step_Down_Timer(IN := FALSE);
    
    IF Step_Up_Timer.Q THEN
        Best_Step := 0;
        Min_Cycles := 16#FFFFFFFF;
        
